PTP {X 66.600,Y -280.193,Z 129.598,A 103.371,B 90.000,C 0.000}
PTP {X 62.438,Y -262.681,Z 129.598,A 103.371,B 90.000,C 0.000}
PTP {X 62.202,Y -262.737,Z 133.786,A 103.319,B 90.000,C 0.000}
PTP {X 66.349,Y -280.253,Z 133.786,A 103.319,B 90.000,C 0.000}
WAIT SEC 2
RET=EKI_SetBool("oxy","torchState",TRUE)
RET = EKI_Send("oxy","torchState")
LIN {X 66.809,Y -282.199,Z 133.786,A 103.319,B 90.000,C 0.000} C_DIS
LIN {X 67.031,Y -282.147,Z 133.851,A 103.364,B 90.000,C 0.000} C_DIS
LIN {X 67.040,Y -282.145,Z 134.927,A 103.366,B 90.000,C 0.000} C_DIS
LIN {X 67.058,Y -282.140,Z 135.029,A 103.370,B 90.000,C 0.000} C_DIS
LIN {X 67.027,Y -282.148,Z 135.471,A 103.363,B 90.000,C 0.000} C_DIS
LIN {X 66.883,Y -282.182,Z 135.935,A 103.334,B 90.000,C 0.000} C_DIS
LIN {X 64.447,Y -282.742,Z 135.913,A 102.840,B 90.000,C 0.000} C_DIS
LIN {X 62.008,Y -283.292,Z 135.871,A 102.346,B 90.000,C 0.000} C_DIS
LIN {X 60.171,Y -283.689,Z 135.751,A 101.975,B 90.000,C 0.000} C_DIS
LIN {X 60.206,Y -283.682,Z 133.837,A 101.982,B 90.000,C 0.000} C_DIS
LIN {X 60.321,Y -283.657,Z 133.653,A 102.005,B 90.000,C 0.000} C_DIS
LIN {X 60.398,Y -283.641,Z 133.605,A 102.021,B 90.000,C 0.000} C_DIS
LIN {X 60.945,Y -283.524,Z 133.589,A 102.131,B 90.000,C 0.000} C_DIS
LIN {X 61.019,Y -283.508,Z 133.573,A 102.146,B 90.000,C 0.000} C_DIS
LIN {X 63.459,Y -282.971,Z 133.658,A 102.640,B 90.000,C 0.000} C_DIS
LIN {X 63.947,Y -282.862,Z 133.676,A 102.739,B 90.000,C 0.000} C_DIS
LIN {X 64.010,Y -282.847,Z 133.664,A 102.752,B 90.000,C 0.000} C_DIS
LIN {X 65.452,Y -282.517,Z 133.698,A 103.044,B 90.000,C 0.000} C_DIS
LIN {X 65.509,Y -282.504,Z 133.682,A 103.055,B 90.000,C 0.000} C_DIS
LIN {X 66.809,Y -282.199,Z 133.786,A 103.319,B 90.000,C 0.000} C_DIS
RET=EKI_SetBool("oxy","torchState",FALSE)
RET = EKI_Send("oxy","torchState")
PTP {X 66.349,Y -280.253,Z 133.786,A 103.319,B 90.000,C 0.000}
PTP {X 62.202,Y -262.737,Z 133.786,A 103.319,B 90.000,C 0.000}
PTP {X 62.126,Y -262.755,Z 137.889,A 103.303,B 90.000,C 0.000}
PTP {X 66.268,Y -280.272,Z 137.889,A 103.303,B 90.000,C 0.000}
WAIT SEC 2
RET=EKI_SetBool("oxy","torchState",TRUE)
RET = EKI_Send("oxy","torchState")
LIN {X 66.728,Y -282.219,Z 137.889,A 103.303,B 90.000,C 0.000} C_DIS
LIN {X 66.797,Y -282.202,Z 138.015,A 103.317,B 90.000,C 0.000} C_DIS
LIN {X 66.769,Y -282.209,Z 139.898,A 103.311,B 90.000,C 0.000} C_DIS
LIN {X 66.664,Y -282.234,Z 140.107,A 103.290,B 90.000,C 0.000} C_DIS
LIN {X 65.640,Y -282.474,Z 140.148,A 103.082,B 90.000,C 0.000} C_DIS
LIN {X 65.555,Y -282.493,Z 140.162,A 103.065,B 90.000,C 0.000} C_DIS
LIN {X 63.119,Y -283.046,Z 140.069,A 102.571,B 90.000,C 0.000} C_DIS
LIN {X 60.679,Y -283.581,Z 139.983,A 102.078,B 90.000,C 0.000} C_DIS
LIN {X 60.222,Y -283.678,Z 139.925,A 101.985,B 90.000,C 0.000} C_DIS
LIN {X 60.149,Y -283.694,Z 139.106,A 101.971,B 90.000,C 0.000} C_DIS
LIN {X 60.192,Y -283.685,Z 138.004,A 101.979,B 90.000,C 0.000} C_DIS
LIN {X 60.238,Y -283.675,Z 137.718,A 101.989,B 90.000,C 0.000} C_DIS
LIN {X 62.449,Y -283.196,Z 137.774,A 102.436,B 90.000,C 0.000} C_DIS
LIN {X 62.511,Y -283.183,Z 137.749,A 102.448,B 90.000,C 0.000} C_DIS
LIN {X 62.630,Y -283.156,Z 137.723,A 102.472,B 90.000,C 0.000} C_DIS
LIN {X 65.064,Y -282.605,Z 137.854,A 102.965,B 90.000,C 0.000} C_DIS
LIN {X 65.785,Y -282.440,Z 137.892,A 103.111,B 90.000,C 0.000} C_DIS
LIN {X 65.895,Y -282.414,Z 137.874,A 103.134,B 90.000,C 0.000} C_DIS
LIN {X 66.728,Y -282.219,Z 137.889,A 103.303,B 90.000,C 0.000} C_DIS
RET=EKI_SetBool("oxy","torchState",FALSE)
RET = EKI_Send("oxy","torchState")
PTP {X 66.268,Y -280.272,Z 137.889,A 103.303,B 90.000,C 0.000}
PTP {X 62.126,Y -262.755,Z 137.889,A 103.303,B 90.000,C 0.000}
PTP {X 63.167,Y -262.507,Z 145.772,A 103.530,B 90.000,C 0.000}
PTP {X 67.378,Y -280.008,Z 145.772,A 103.530,B 90.000,C 0.000}
WAIT SEC 2
RET=EKI_SetBool("oxy","torchState",TRUE)
RET = EKI_Send("oxy","torchState")
LIN {X 67.846,Y -281.952,Z 145.772,A 103.530,B 90.000,C 0.000} C_DIS
LIN {X 67.709,Y -281.985,Z 145.810,A 103.502,B 90.000,C 0.000} C_DIS
LIN {X 67.614,Y -282.008,Z 145.931,A 103.483,B 90.000,C 0.000} C_DIS
LIN {X 67.474,Y -282.041,Z 147.023,A 103.454,B 90.000,C 0.000} C_DIS
LIN {X 67.502,Y -282.035,Z 147.081,A 103.460,B 90.000,C 0.000} C_DIS
LIN {X 67.529,Y -282.028,Z 147.194,A 103.465,B 90.000,C 0.000} C_DIS
LIN {X 67.438,Y -282.050,Z 149.692,A 103.447,B 90.000,C 0.000} C_DIS
LIN {X 67.377,Y -282.064,Z 152.191,A 103.435,B 90.000,C 0.000} C_DIS
LIN {X 67.312,Y -282.080,Z 153.552,A 103.421,B 90.000,C 0.000} C_DIS
LIN {X 67.335,Y -282.075,Z 153.680,A 103.426,B 90.000,C 0.000} C_DIS
LIN {X 67.359,Y -282.069,Z 153.744,A 103.431,B 90.000,C 0.000} C_DIS
LIN {X 67.267,Y -282.091,Z 156.242,A 103.412,B 90.000,C 0.000} C_DIS
LIN {X 67.200,Y -282.107,Z 157.545,A 103.399,B 90.000,C 0.000} C_DIS
LIN {X 67.251,Y -282.094,Z 157.665,A 103.409,B 90.000,C 0.000} C_DIS
LIN {X 67.142,Y -282.120,Z 159.596,A 103.387,B 90.000,C 0.000} C_DIS
LIN {X 67.193,Y -282.108,Z 159.718,A 103.397,B 90.000,C 0.000} C_DIS
LIN {X 67.089,Y -282.133,Z 161.522,A 103.376,B 90.000,C 0.000} C_DIS
LIN {X 67.066,Y -282.138,Z 163.614,A 103.371,B 90.000,C 0.000} C_DIS
LIN {X 67.082,Y -282.135,Z 163.700,A 103.375,B 90.000,C 0.000} C_DIS
LIN {X 66.977,Y -282.160,Z 165.512,A 103.353,B 90.000,C 0.000} C_DIS
LIN {X 67.026,Y -282.148,Z 165.700,A 103.363,B 90.000,C 0.000} C_DIS
LIN {X 66.921,Y -282.173,Z 167.562,A 103.342,B 90.000,C 0.000} C_DIS
LIN {X 66.950,Y -282.166,Z 167.620,A 103.348,B 90.000,C 0.000} C_DIS
LIN {X 66.977,Y -282.160,Z 167.720,A 103.353,B 90.000,C 0.000} C_DIS
LIN {X 66.865,Y -282.186,Z 169.553,A 103.331,B 90.000,C 0.000} C_DIS
LIN {X 66.919,Y -282.173,Z 169.669,A 103.342,B 90.000,C 0.000} C_DIS
LIN {X 66.814,Y -282.198,Z 171.481,A 103.320,B 90.000,C 0.000} C_DIS
LIN {X 66.838,Y -282.193,Z 171.575,A 103.325,B 90.000,C 0.000} C_DIS
LIN {X 66.861,Y -282.187,Z 171.729,A 103.330,B 90.000,C 0.000} C_DIS
LIN {X 66.757,Y -282.212,Z 173.475,A 103.309,B 90.000,C 0.000} C_DIS
LIN {X 66.804,Y -282.201,Z 173.665,A 103.318,B 90.000,C 0.000} C_DIS
LIN {X 66.702,Y -282.225,Z 175.522,A 103.298,B 90.000,C 0.000} C_DIS
LIN {X 66.727,Y -282.219,Z 175.585,A 103.303,B 90.000,C 0.000} C_DIS
LIN {X 66.753,Y -282.213,Z 175.702,A 103.308,B 90.000,C 0.000} C_DIS
LIN {X 66.647,Y -282.238,Z 177.513,A 103.286,B 90.000,C 0.000} C_DIS
LIN {X 66.696,Y -282.226,Z 177.638,A 103.296,B 90.000,C 0.000} C_DIS
LIN {X 66.604,Y -282.248,Z 180.136,A 103.278,B 90.000,C 0.000} C_DIS
LIN {X 66.541,Y -282.263,Z 182.635,A 103.265,B 90.000,C 0.000} C_DIS
LIN {X 66.482,Y -282.277,Z 183.486,A 103.253,B 90.000,C 0.000} C_DIS
LIN {X 66.505,Y -282.271,Z 183.551,A 103.258,B 90.000,C 0.000} C_DIS
LIN {X 66.530,Y -282.265,Z 183.673,A 103.263,B 90.000,C 0.000} C_DIS
LIN {X 66.435,Y -282.288,Z 186.171,A 103.243,B 90.000,C 0.000} C_DIS
LIN {X 66.371,Y -282.303,Z 188.670,A 103.230,B 90.000,C 0.000} C_DIS
LIN {X 66.301,Y -282.319,Z 191.169,A 103.216,B 90.000,C 0.000} C_DIS
LIN {X 66.233,Y -282.335,Z 193.668,A 103.202,B 90.000,C 0.000} C_DIS
LIN {X 66.164,Y -282.351,Z 196.167,A 103.188,B 90.000,C 0.000} C_DIS
LIN {X 66.094,Y -282.368,Z 198.666,A 103.174,B 90.000,C 0.000} C_DIS
LIN {X 66.026,Y -282.384,Z 201.165,A 103.160,B 90.000,C 0.000} C_DIS
LIN {X 65.962,Y -282.399,Z 203.664,A 103.147,B 90.000,C 0.000} C_DIS
LIN {X 65.872,Y -282.420,Z 205.953,A 103.129,B 90.000,C 0.000} C_DIS
LIN {X 65.895,Y -282.414,Z 206.081,A 103.134,B 90.000,C 0.000} C_DIS
LIN {X 65.919,Y -282.409,Z 206.145,A 103.139,B 90.000,C 0.000} C_DIS
LIN {X 65.815,Y -282.433,Z 207.949,A 103.118,B 90.000,C 0.000} C_DIS
LIN {X 65.778,Y -282.442,Z 209.438,A 103.110,B 90.000,C 0.000} C_DIS
LIN {X 65.893,Y -282.415,Z 210.148,A 103.133,B 90.000,C 0.000} C_DIS
LIN {X 66.114,Y -282.363,Z 210.265,A 103.178,B 90.000,C 0.000} C_DIS
LIN {X 68.542,Y -281.784,Z 210.399,A 103.671,B 90.000,C 0.000} C_DIS
LIN {X 70.968,Y -281.181,Z 210.381,A 104.165,B 90.000,C 0.000} C_DIS
LIN {X 72.559,Y -280.776,Z 210.270,A 104.489,B 90.000,C 0.000} C_DIS
LIN {X 73.021,Y -280.656,Z 210.199,A 104.584,B 90.000,C 0.000} C_DIS
LIN {X 73.200,Y -280.610,Z 210.143,A 104.620,B 90.000,C 0.000} C_DIS
LIN {X 75.002,Y -280.133,Z 209.853,A 104.989,B 90.000,C 0.000} C_DIS
LIN {X 75.137,Y -280.097,Z 209.840,A 105.016,B 90.000,C 0.000} C_DIS
LIN {X 76.430,Y -279.747,Z 209.490,A 105.281,B 90.000,C 0.000} C_DIS
LIN {X 76.539,Y -279.717,Z 209.479,A 105.303,B 90.000,C 0.000} C_DIS
LIN {X 76.649,Y -279.687,Z 209.442,A 105.326,B 90.000,C 0.000} C_DIS
LIN {X 76.707,Y -279.671,Z 209.412,A 105.338,B 90.000,C 0.000} C_DIS
LIN {X 77.910,Y -279.338,Z 209.194,A 105.584,B 90.000,C 0.000} C_DIS
LIN {X 78.896,Y -279.062,Z 208.865,A 105.787,B 90.000,C 0.000} C_DIS
LIN {X 79.006,Y -279.031,Z 208.853,A 105.809,B 90.000,C 0.000} C_DIS
LIN {X 79.115,Y -279.000,Z 208.815,A 105.832,B 90.000,C 0.000} C_DIS
LIN {X 79.827,Y -278.797,Z 208.658,A 105.978,B 90.000,C 0.000} C_DIS
LIN {X 79.936,Y -278.766,Z 208.645,A 106.000,B 90.000,C 0.000} C_DIS
LIN {X 80.538,Y -278.592,Z 208.403,A 106.124,B 90.000,C 0.000} C_DIS
LIN {X 80.647,Y -278.561,Z 208.374,A 106.146,B 90.000,C 0.000} C_DIS
LIN {X 80.756,Y -278.529,Z 208.362,A 106.169,B 90.000,C 0.000} C_DIS
LIN {X 81.548,Y -278.298,Z 208.093,A 106.332,B 90.000,C 0.000} C_DIS
LIN {X 81.630,Y -278.274,Z 208.080,A 106.349,B 90.000,C 0.000} C_DIS
LIN {X 82.830,Y -277.919,Z 207.617,A 106.596,B 90.000,C 0.000} C_DIS
LIN {X 83.757,Y -277.641,Z 207.332,A 106.787,B 90.000,C 0.000} C_DIS
LIN {X 83.975,Y -277.576,Z 207.294,A 106.832,B 90.000,C 0.000} C_DIS
LIN {X 84.846,Y -277.311,Z 206.990,A 107.012,B 90.000,C 0.000} C_DIS
LIN {X 85.063,Y -277.244,Z 206.951,A 107.057,B 90.000,C 0.000} C_DIS
LIN {X 86.613,Y -276.764,Z 206.308,A 107.377,B 90.000,C 0.000} C_DIS
LIN {X 86.697,Y -276.737,Z 206.283,A 107.395,B 90.000,C 0.000} C_DIS
LIN {X 87.703,Y -276.420,Z 205.797,A 107.603,B 90.000,C 0.000} C_DIS
LIN {X 88.687,Y -276.106,Z 205.372,A 107.807,B 90.000,C 0.000} C_DIS
LIN {X 88.808,Y -276.067,Z 205.284,A 107.833,B 90.000,C 0.000} C_DIS
LIN {X 89.188,Y -275.945,Z 205.105,A 107.911,B 90.000,C 0.000} C_DIS
LIN {X 89.296,Y -275.910,Z 205.067,A 107.934,B 90.000,C 0.000} C_DIS
LIN {X 89.823,Y -275.739,Z 204.794,A 108.043,B 90.000,C 0.000} C_DIS
LIN {X 90.663,Y -275.464,Z 204.379,A 108.218,B 90.000,C 0.000} C_DIS
LIN {X 92.554,Y -274.834,Z 202.870,A 108.612,B 90.000,C 0.000} C_DIS
LIN {X 93.451,Y -274.530,Z 202.156,A 108.799,B 90.000,C 0.000} C_DIS
LIN {X 93.559,Y -274.494,Z 201.985,A 108.821,B 90.000,C 0.000} C_DIS
LIN {X 94.606,Y -274.134,Z 200.990,A 109.040,B 90.000,C 0.000} C_DIS
LIN {X 94.818,Y -274.061,Z 200.829,A 109.084,B 90.000,C 0.000} C_DIS
LIN {X 94.853,Y -274.049,Z 200.808,A 109.092,B 90.000,C 0.000} C_DIS
LIN {X 95.087,Y -273.968,Z 200.545,A 109.140,B 90.000,C 0.000} C_DIS
LIN {X 95.122,Y -273.956,Z 200.519,A 109.148,B 90.000,C 0.000} C_DIS
LIN {X 96.142,Y -273.600,Z 199.308,A 109.361,B 90.000,C 0.000} C_DIS
LIN {X 96.196,Y -273.581,Z 199.282,A 109.373,B 90.000,C 0.000} C_DIS
LIN {X 96.303,Y -273.543,Z 199.169,A 109.395,B 90.000,C 0.000} C_DIS
LIN {X 96.357,Y -273.524,Z 199.141,A 109.406,B 90.000,C 0.000} C_DIS
LIN {X 97.431,Y -273.143,Z 198.002,A 109.631,B 90.000,C 0.000} C_DIS
LIN {X 97.483,Y -273.125,Z 197.926,A 109.642,B 90.000,C 0.000} C_DIS
LIN {X 97.808,Y -273.008,Z 197.547,A 109.711,B 90.000,C 0.000} C_DIS
LIN {X 98.019,Y -272.933,Z 197.324,A 109.755,B 90.000,C 0.000} C_DIS
LIN {X 98.099,Y -272.904,Z 197.263,A 109.772,B 90.000,C 0.000} C_DIS
LIN {X 98.179,Y -272.875,Z 197.185,A 109.788,B 90.000,C 0.000} C_DIS
LIN {X 98.447,Y -272.779,Z 196.822,A 109.845,B 90.000,C 0.000} C_DIS
LIN {X 98.607,Y -272.721,Z 196.691,A 109.878,B 90.000,C 0.000} C_DIS
LIN {X 99.051,Y -272.560,Z 196.054,A 109.972,B 90.000,C 0.000} C_DIS
LIN {X 99.196,Y -272.507,Z 195.893,A 110.002,B 90.000,C 0.000} C_DIS
LIN {X 99.262,Y -272.483,Z 195.758,A 110.016,B 90.000,C 0.000} C_DIS
LIN {X 99.556,Y -272.376,Z 195.354,A 110.078,B 90.000,C 0.000} C_DIS
LIN {X 99.623,Y -272.351,Z 195.227,A 110.092,B 90.000,C 0.000} C_DIS
LIN {X 99.883,Y -272.256,Z 194.840,A 110.147,B 90.000,C 0.000} C_DIS
LIN {X 99.968,Y -272.225,Z 194.655,A 110.164,B 90.000,C 0.000} C_DIS
LIN {X 100.104,Y -272.175,Z 194.472,A 110.193,B 90.000,C 0.000} C_DIS
LIN {X 100.380,Y -272.073,Z 194.019,A 110.251,B 90.000,C 0.000} C_DIS
LIN {X 100.452,Y -272.047,Z 193.834,A 110.267,B 90.000,C 0.000} C_DIS
LIN {X 101.164,Y -271.783,Z 192.678,A 110.416,B 90.000,C 0.000} C_DIS
LIN {X 101.248,Y -271.751,Z 192.493,A 110.434,B 90.000,C 0.000} C_DIS
LIN {X 101.331,Y -271.721,Z 192.369,A 110.452,B 90.000,C 0.000} C_DIS
LIN {X 101.568,Y -271.632,Z 191.936,A 110.502,B 90.000,C 0.000} C_DIS
LIN {X 101.758,Y -271.561,Z 191.510,A 110.542,B 90.000,C 0.000} C_DIS
LIN {X 101.917,Y -271.501,Z 191.230,A 110.575,B 90.000,C 0.000} C_DIS
LIN {X 101.990,Y -271.474,Z 191.048,A 110.591,B 90.000,C 0.000} C_DIS
LIN {X 102.290,Y -271.361,Z 190.459,A 110.654,B 90.000,C 0.000} C_DIS
LIN {X 102.665,Y -271.219,Z 189.752,A 110.733,B 90.000,C 0.000} C_DIS
LIN {X 102.929,Y -271.119,Z 189.330,A 110.789,B 90.000,C 0.000} C_DIS
LIN {X 103.194,Y -271.018,Z 188.842,A 110.845,B 90.000,C 0.000} C_DIS
LIN {X 103.731,Y -270.813,Z 187.875,A 110.959,B 90.000,C 0.000} C_DIS
LIN {X 104.098,Y -270.673,Z 187.190,A 111.036,B 90.000,C 0.000} C_DIS
LIN {X 104.287,Y -270.600,Z 186.773,A 111.076,B 90.000,C 0.000} C_DIS
LIN {X 105.306,Y -270.205,Z 184.524,A 111.292,B 90.000,C 0.000} C_DIS
LIN {X 106.047,Y -269.915,Z 182.154,A 111.449,B 90.000,C 0.000} C_DIS
LIN {X 106.672,Y -269.668,Z 179.747,A 111.582,B 90.000,C 0.000} C_DIS
LIN {X 106.947,Y -269.560,Z 178.502,A 111.641,B 90.000,C 0.000} C_DIS
LIN {X 107.012,Y -269.534,Z 178.401,A 111.654,B 90.000,C 0.000} C_DIS
LIN {X 107.641,Y -269.283,Z 175.995,A 111.788,B 90.000,C 0.000} C_DIS
LIN {X 108.204,Y -269.057,Z 173.569,A 111.908,B 90.000,C 0.000} C_DIS
LIN {X 108.758,Y -268.834,Z 171.142,A 112.026,B 90.000,C 0.000} C_DIS
LIN {X 109.297,Y -268.615,Z 168.710,A 112.141,B 90.000,C 0.000} C_DIS
LIN {X 109.764,Y -268.425,Z 166.262,A 112.241,B 90.000,C 0.000} C_DIS
LIN {X 110.124,Y -268.277,Z 163.793,A 112.317,B 90.000,C 0.000} C_DIS
LIN {X 110.419,Y -268.156,Z 161.313,A 112.380,B 90.000,C 0.000} C_DIS
LIN {X 110.734,Y -268.026,Z 158.836,A 112.448,B 90.000,C 0.000} C_DIS
LIN {X 111.105,Y -267.873,Z 156.369,A 112.527,B 90.000,C 0.000} C_DIS
LIN {X 111.493,Y -267.711,Z 153.905,A 112.610,B 90.000,C 0.000} C_DIS
LIN {X 111.867,Y -267.555,Z 151.438,A 112.690,B 90.000,C 0.000} C_DIS
LIN {X 111.944,Y -267.523,Z 150.914,A 112.707,B 90.000,C 0.000} C_DIS
LIN {X 111.866,Y -267.556,Z 150.619,A 112.690,B 90.000,C 0.000} C_DIS
LIN {X 111.637,Y -267.651,Z 150.611,A 112.641,B 90.000,C 0.000} C_DIS
LIN {X 111.312,Y -267.787,Z 150.818,A 112.571,B 90.000,C 0.000} C_DIS
LIN {X 110.388,Y -268.169,Z 152.148,A 112.374,B 90.000,C 0.000} C_DIS
LIN {X 110.323,Y -268.196,Z 152.283,A 112.360,B 90.000,C 0.000} C_DIS
LIN {X 110.033,Y -268.315,Z 152.687,A 112.298,B 90.000,C 0.000} C_DIS
LIN {X 109.967,Y -268.342,Z 152.823,A 112.284,B 90.000,C 0.000} C_DIS
LIN {X 109.888,Y -268.374,Z 152.884,A 112.267,B 90.000,C 0.000} C_DIS
LIN {X 109.809,Y -268.406,Z 152.967,A 112.250,B 90.000,C 0.000} C_DIS
LIN {X 109.230,Y -268.643,Z 153.798,A 112.127,B 90.000,C 0.000} C_DIS
LIN {X 108.492,Y -268.942,Z 154.770,A 111.969,B 90.000,C 0.000} C_DIS
LIN {X 108.452,Y -268.958,Z 154.799,A 111.961,B 90.000,C 0.000} C_DIS
LIN {X 108.344,Y -269.001,Z 154.853,A 111.938,B 90.000,C 0.000} C_DIS
LIN {X 108.308,Y -269.015,Z 154.932,A 111.930,B 90.000,C 0.000} C_DIS
LIN {X 107.700,Y -269.260,Z 155.660,A 111.801,B 90.000,C 0.000} C_DIS
LIN {X 107.466,Y -269.353,Z 155.857,A 111.751,B 90.000,C 0.000} C_DIS
LIN {X 107.013,Y -269.534,Z 156.459,A 111.654,B 90.000,C 0.000} C_DIS
LIN {X 106.880,Y -269.586,Z 156.582,A 111.626,B 90.000,C 0.000} C_DIS
LIN {X 106.245,Y -269.837,Z 157.322,A 111.492,B 90.000,C 0.000} C_DIS
LIN {X 106.166,Y -269.868,Z 157.383,A 111.475,B 90.000,C 0.000} C_DIS
LIN {X 105.958,Y -269.950,Z 157.606,A 111.430,B 90.000,C 0.000} C_DIS
LIN {X 104.629,Y -270.468,Z 159.264,A 111.149,B 90.000,C 0.000} C_DIS
LIN {X 104.523,Y -270.509,Z 159.301,A 111.126,B 90.000,C 0.000} C_DIS
LIN {X 104.416,Y -270.550,Z 159.484,A 111.104,B 90.000,C 0.000} C_DIS
LIN {X 104.204,Y -270.632,Z 159.654,A 111.059,B 90.000,C 0.000} C_DIS
LIN {X 104.098,Y -270.673,Z 159.837,A 111.036,B 90.000,C 0.000} C_DIS
LIN {X 104.045,Y -270.693,Z 159.853,A 111.025,B 90.000,C 0.000} C_DIS
LIN {X 103.992,Y -270.713,Z 159.879,A 111.014,B 90.000,C 0.000} C_DIS
LIN {X 103.939,Y -270.734,Z 159.939,A 111.003,B 90.000,C 0.000} C_DIS
LIN {X 102.916,Y -271.124,Z 160.863,A 110.786,B 90.000,C 0.000} C_DIS
LIN {X 102.761,Y -271.183,Z 160.963,A 110.753,B 90.000,C 0.000} C_DIS
LIN {X 101.118,Y -271.800,Z 162.344,A 110.407,B 90.000,C 0.000} C_DIS
LIN {X 101.011,Y -271.840,Z 162.370,A 110.384,B 90.000,C 0.000} C_DIS
LIN {X 99.164,Y -272.519,Z 163.912,A 109.996,B 90.000,C 0.000} C_DIS
LIN {X 97.915,Y -272.970,Z 164.946,A 109.733,B 90.000,C 0.000} C_DIS
LIN {X 96.893,Y -273.334,Z 165.569,A 109.519,B 90.000,C 0.000} C_DIS
LIN {X 96.679,Y -273.410,Z 165.629,A 109.474,B 90.000,C 0.000} C_DIS
LIN {X 96.303,Y -273.543,Z 165.812,A 109.395,B 90.000,C 0.000} C_DIS
LIN {X 96.088,Y -273.618,Z 165.859,A 109.350,B 90.000,C 0.000} C_DIS
LIN {X 95.713,Y -273.750,Z 166.028,A 109.271,B 90.000,C 0.000} C_DIS
LIN {X 95.498,Y -273.825,Z 166.067,A 109.226,B 90.000,C 0.000} C_DIS
LIN {X 94.630,Y -274.126,Z 166.389,A 109.045,B 90.000,C 0.000} C_DIS
LIN {X 93.080,Y -274.656,Z 166.682,A 108.721,B 90.000,C 0.000} C_DIS
LIN {X 93.001,Y -274.683,Z 166.718,A 108.705,B 90.000,C 0.000} C_DIS
LIN {X 92.699,Y -274.785,Z 166.760,A 108.642,B 90.000,C 0.000} C_DIS
LIN {X 92.626,Y -274.810,Z 166.790,A 108.627,B 90.000,C 0.000} C_DIS
LIN {X 91.350,Y -275.236,Z 166.921,A 108.361,B 90.000,C 0.000} C_DIS
LIN {X 90.329,Y -275.573,Z 166.912,A 108.148,B 90.000,C 0.000} C_DIS
LIN {X 90.217,Y -275.610,Z 166.966,A 108.125,B 90.000,C 0.000} C_DIS
LIN {X 87.844,Y -276.375,Z 166.775,A 107.633,B 90.000,C 0.000} C_DIS
LIN {X 87.119,Y -276.605,Z 166.677,A 107.482,B 90.000,C 0.000} C_DIS
LIN {X 84.832,Y -277.315,Z 165.959,A 107.009,B 90.000,C 0.000} C_DIS
LIN {X 82.557,Y -278.000,Z 165.182,A 106.540,B 90.000,C 0.000} C_DIS
LIN {X 80.348,Y -278.647,Z 164.206,A 106.085,B 90.000,C 0.000} C_DIS
LIN {X 79.018,Y -279.027,Z 163.487,A 105.812,B 90.000,C 0.000} C_DIS
LIN {X 78.732,Y -279.108,Z 163.351,A 105.753,B 90.000,C 0.000} C_DIS
LIN {X 77.702,Y -279.397,Z 162.449,A 105.542,B 90.000,C 0.000} C_DIS
LIN {X 77.129,Y -279.555,Z 161.793,A 105.424,B 90.000,C 0.000} C_DIS
LIN {X 76.943,Y -279.606,Z 161.674,A 105.386,B 90.000,C 0.000} C_DIS
LIN {X 75.441,Y -280.015,Z 160.166,A 105.078,B 90.000,C 0.000} C_DIS
LIN {X 74.857,Y -280.172,Z 159.269,A 104.959,B 90.000,C 0.000} C_DIS
LIN {X 74.741,Y -280.203,Z 158.962,A 104.935,B 90.000,C 0.000} C_DIS
LIN {X 74.452,Y -280.280,Z 158.354,A 104.876,B 90.000,C 0.000} C_DIS
LIN {X 74.402,Y -280.293,Z 158.289,A 104.866,B 90.000,C 0.000} C_DIS
LIN {X 74.351,Y -280.307,Z 158.061,A 104.855,B 90.000,C 0.000} C_DIS
LIN {X 74.147,Y -280.361,Z 157.610,A 104.814,B 90.000,C 0.000} C_DIS
LIN {X 74.129,Y -280.366,Z 157.525,A 104.810,B 90.000,C 0.000} C_DIS
LIN {X 73.627,Y -280.498,Z 156.152,A 104.708,B 90.000,C 0.000} C_DIS
LIN {X 73.751,Y -280.465,Z 156.076,A 104.733,B 90.000,C 0.000} C_DIS
LIN {X 74.007,Y -280.398,Z 156.226,A 104.785,B 90.000,C 0.000} C_DIS
LIN {X 74.243,Y -280.336,Z 156.451,A 104.833,B 90.000,C 0.000} C_DIS
LIN {X 74.452,Y -280.280,Z 156.750,A 104.876,B 90.000,C 0.000} C_DIS
LIN {X 74.516,Y -280.263,Z 156.810,A 104.889,B 90.000,C 0.000} C_DIS
LIN {X 74.546,Y -280.255,Z 156.845,A 104.895,B 90.000,C 0.000} C_DIS
LIN {X 75.606,Y -279.971,Z 158.296,A 105.112,B 90.000,C 0.000} C_DIS
LIN {X 76.808,Y -279.644,Z 159.541,A 105.358,B 90.000,C 0.000} C_DIS
LIN {X 77.227,Y -279.528,Z 159.825,A 105.444,B 90.000,C 0.000} C_DIS
LIN {X 77.394,Y -279.482,Z 159.967,A 105.479,B 90.000,C 0.000} C_DIS
LIN {X 77.606,Y -279.423,Z 160.109,A 105.522,B 90.000,C 0.000} C_DIS
LIN {X 77.691,Y -279.399,Z 160.195,A 105.539,B 90.000,C 0.000} C_DIS
LIN {X 77.748,Y -279.384,Z 160.280,A 105.551,B 90.000,C 0.000} C_DIS
LIN {X 78.369,Y -279.210,Z 160.753,A 105.679,B 90.000,C 0.000} C_DIS
LIN {X 78.515,Y -279.169,Z 160.906,A 105.708,B 90.000,C 0.000} C_DIS
LIN {X 78.639,Y -279.134,Z 160.964,A 105.734,B 90.000,C 0.000} C_DIS
LIN {X 79.151,Y -278.990,Z 161.333,A 105.839,B 90.000,C 0.000} C_DIS
LIN {X 80.846,Y -278.503,Z 162.328,A 106.187,B 90.000,C 0.000} C_DIS
LIN {X 80.920,Y -278.481,Z 162.383,A 106.203,B 90.000,C 0.000} C_DIS
LIN {X 81.866,Y -278.205,Z 162.810,A 106.397,B 90.000,C 0.000} C_DIS
LIN {X 82.273,Y -278.085,Z 163.047,A 106.481,B 90.000,C 0.000} C_DIS
LIN {X 82.447,Y -278.033,Z 163.125,A 106.517,B 90.000,C 0.000} C_DIS
LIN {X 84.030,Y -277.559,Z 163.866,A 106.843,B 90.000,C 0.000} C_DIS
LIN {X 86.363,Y -276.840,Z 164.401,A 107.326,B 90.000,C 0.000} C_DIS
LIN {X 87.752,Y -276.405,Z 164.640,A 107.613,B 90.000,C 0.000} C_DIS
LIN {X 90.131,Y -275.637,Z 164.640,A 108.107,B 90.000,C 0.000} C_DIS
LIN {X 91.761,Y -275.100,Z 164.513,A 108.446,B 90.000,C 0.000} C_DIS
LIN {X 91.836,Y -275.075,Z 164.484,A 108.462,B 90.000,C 0.000} C_DIS
LIN {X 93.171,Y -274.626,Z 164.264,A 108.740,B 90.000,C 0.000} C_DIS
LIN {X 93.292,Y -274.584,Z 164.199,A 108.766,B 90.000,C 0.000} C_DIS
LIN {X 93.380,Y -274.555,Z 164.172,A 108.784,B 90.000,C 0.000} C_DIS
LIN {X 93.777,Y -274.419,Z 164.099,A 108.867,B 90.000,C 0.000} C_DIS
LIN {X 95.444,Y -273.844,Z 163.519,A 109.215,B 90.000,C 0.000} C_DIS
LIN {X 95.511,Y -273.820,Z 163.468,A 109.229,B 90.000,C 0.000} C_DIS
LIN {X 96.402,Y -273.508,Z 162.997,A 109.416,B 90.000,C 0.000} C_DIS
LIN {X 96.469,Y -273.485,Z 162.986,A 109.430,B 90.000,C 0.000} C_DIS
LIN {X 96.989,Y -273.301,Z 162.727,A 109.539,B 90.000,C 0.000} C_DIS
LIN {X 97.342,Y -273.175,Z 162.596,A 109.613,B 90.000,C 0.000} C_DIS
LIN {X 97.376,Y -273.163,Z 162.565,A 109.620,B 90.000,C 0.000} C_DIS
LIN {X 97.469,Y -273.129,Z 162.499,A 109.640,B 90.000,C 0.000} C_DIS
LIN {X 97.978,Y -272.947,Z 162.272,A 109.746,B 90.000,C 0.000} C_DIS
LIN {X 98.458,Y -272.775,Z 161.955,A 109.847,B 90.000,C 0.000} C_DIS
LIN {X 98.643,Y -272.708,Z 161.852,A 109.886,B 90.000,C 0.000} C_DIS
LIN {X 98.926,Y -272.605,Z 161.646,A 109.945,B 90.000,C 0.000} C_DIS
LIN {X 99.013,Y -272.574,Z 161.546,A 109.964,B 90.000,C 0.000} C_DIS
LIN {X 99.249,Y -272.488,Z 161.371,A 110.013,B 90.000,C 0.000} C_DIS
LIN {X 99.946,Y -272.233,Z 160.721,A 110.160,B 90.000,C 0.000} C_DIS
LIN {X 100.102,Y -272.176,Z 160.521,A 110.193,B 90.000,C 0.000} C_DIS
LIN {X 101.700,Y -271.583,Z 159.072,A 110.529,B 90.000,C 0.000} C_DIS
LIN {X 101.811,Y -271.541,Z 158.998,A 110.553,B 90.000,C 0.000} C_DIS
LIN {X 103.534,Y -270.889,Z 157.309,A 110.917,B 90.000,C 0.000} C_DIS
LIN {X 104.204,Y -270.632,Z 156.381,A 111.059,B 90.000,C 0.000} C_DIS
LIN {X 104.257,Y -270.611,Z 156.326,A 111.070,B 90.000,C 0.000} C_DIS
LIN {X 104.310,Y -270.591,Z 156.302,A 111.081,B 90.000,C 0.000} C_DIS
LIN {X 104.894,Y -270.365,Z 155.561,A 111.205,B 90.000,C 0.000} C_DIS
LIN {X 104.947,Y -270.344,Z 155.529,A 111.216,B 90.000,C 0.000} C_DIS
LIN {X 105.000,Y -270.324,Z 155.509,A 111.227,B 90.000,C 0.000} C_DIS
LIN {X 106.587,Y -269.702,Z 153.680,A 111.564,B 90.000,C 0.000} C_DIS
LIN {X 107.541,Y -269.323,Z 152.538,A 111.767,B 90.000,C 0.000} C_DIS
LIN {X 107.594,Y -269.302,Z 152.514,A 111.778,B 90.000,C 0.000} C_DIS
LIN {X 107.647,Y -269.281,Z 152.480,A 111.789,B 90.000,C 0.000} C_DIS
LIN {X 108.333,Y -269.005,Z 151.590,A 111.936,B 90.000,C 0.000} C_DIS
LIN {X 108.492,Y -268.942,Z 151.457,A 111.969,B 90.000,C 0.000} C_DIS
LIN {X 108.558,Y -268.915,Z 151.315,A 111.983,B 90.000,C 0.000} C_DIS
LIN {X 109.190,Y -268.659,Z 150.547,A 112.118,B 90.000,C 0.000} C_DIS
LIN {X 109.335,Y -268.600,Z 150.320,A 112.149,B 90.000,C 0.000} C_DIS
LIN {X 109.493,Y -268.535,Z 150.142,A 112.183,B 90.000,C 0.000} C_DIS
LIN {X 110.275,Y -268.215,Z 149.144,A 112.350,B 90.000,C 0.000} C_DIS
LIN {X 110.407,Y -268.161,Z 149.054,A 112.378,B 90.000,C 0.000} C_DIS
LIN {X 110.757,Y -268.017,Z 148.530,A 112.453,B 90.000,C 0.000} C_DIS
LIN {X 110.809,Y -267.995,Z 148.474,A 112.464,B 90.000,C 0.000} C_DIS
LIN {X 110.862,Y -267.973,Z 148.450,A 112.475,B 90.000,C 0.000} C_DIS
LIN {X 111.177,Y -267.843,Z 147.995,A 112.543,B 90.000,C 0.000} C_DIS
LIN {X 111.226,Y -267.822,Z 147.960,A 112.553,B 90.000,C 0.000} C_DIS
LIN {X 111.308,Y -267.788,Z 147.878,A 112.571,B 90.000,C 0.000} C_DIS
LIN {X 111.391,Y -267.754,Z 147.763,A 112.588,B 90.000,C 0.000} C_DIS
LIN {X 112.204,Y -267.414,Z 146.500,A 112.762,B 90.000,C 0.000} C_DIS
LIN {X 113.158,Y -267.012,Z 144.224,A 112.967,B 90.000,C 0.000} C_DIS
LIN {X 113.967,Y -266.667,Z 141.884,A 113.141,B 90.000,C 0.000} C_DIS
LIN {X 114.668,Y -266.367,Z 139.503,A 113.291,B 90.000,C 0.000} C_DIS
LIN {X 115.419,Y -266.042,Z 137.141,A 113.453,B 90.000,C 0.000} C_DIS
LIN {X 116.181,Y -265.710,Z 134.783,A 113.617,B 90.000,C 0.000} C_DIS
LIN {X 116.912,Y -265.390,Z 132.414,A 113.775,B 90.000,C 0.000} C_DIS
LIN {X 117.615,Y -265.079,Z 130.035,A 113.927,B 90.000,C 0.000} C_DIS
LIN {X 118.323,Y -264.763,Z 127.659,A 114.080,B 90.000,C 0.000} C_DIS
LIN {X 119.096,Y -264.416,Z 125.307,A 114.247,B 90.000,C 0.000} C_DIS
LIN {X 119.968,Y -264.022,Z 122.997,A 114.436,B 90.000,C 0.000} C_DIS
LIN {X 120.871,Y -263.610,Z 120.703,A 114.632,B 90.000,C 0.000} C_DIS
LIN {X 121.669,Y -263.242,Z 118.620,A 114.806,B 90.000,C 0.000} C_DIS
LIN {X 121.984,Y -263.097,Z 117.906,A 114.875,B 90.000,C 0.000} C_DIS
LIN {X 122.322,Y -262.940,Z 117.160,A 114.948,B 90.000,C 0.000} C_DIS
LIN {X 123.186,Y -262.536,Z 114.849,A 115.137,B 90.000,C 0.000} C_DIS
LIN {X 124.147,Y -262.083,Z 112.587,A 115.347,B 90.000,C 0.000} C_DIS
LIN {X 124.998,Y -261.678,Z 110.271,A 115.533,B 90.000,C 0.000} C_DIS
LIN {X 125.720,Y -261.332,Z 107.903,A 115.691,B 90.000,C 0.000} C_DIS
LIN {X 126.434,Y -260.988,Z 105.532,A 115.848,B 90.000,C 0.000} C_DIS
LIN {X 127.087,Y -260.670,Z 103.140,A 115.991,B 90.000,C 0.000} C_DIS
LIN {X 127.896,Y -260.274,Z 100.808,A 116.169,B 90.000,C 0.000} C_DIS
LIN {X 128.611,Y -259.921,Z 98.438,A 116.327,B 90.000,C 0.000} C_DIS
LIN {X 129.304,Y -259.577,Z 96.061,A 116.479,B 90.000,C 0.000} C_DIS
LIN {X 129.860,Y -259.300,Z 93.826,A 116.602,B 90.000,C 0.000} C_DIS
LIN {X 129.878,Y -259.291,Z 91.326,A 116.606,B 90.000,C 0.000} C_DIS
LIN {X 129.664,Y -259.398,Z 90.184,A 116.559,B 90.000,C 0.000} C_DIS
LIN {X 129.650,Y -259.405,Z 90.071,A 116.556,B 90.000,C 0.000} C_DIS
LIN {X 129.441,Y -259.509,Z 89.331,A 116.510,B 90.000,C 0.000} C_DIS
LIN {X 129.431,Y -259.514,Z 89.217,A 116.507,B 90.000,C 0.000} C_DIS
LIN {X 129.405,Y -259.527,Z 89.103,A 116.502,B 90.000,C 0.000} C_DIS
LIN {X 128.834,Y -259.811,Z 87.432,A 116.376,B 90.000,C 0.000} C_DIS
LIN {X 128.444,Y -260.004,Z 86.844,A 116.290,B 90.000,C 0.000} C_DIS
LIN {X 127.967,Y -260.239,Z 86.374,A 116.185,B 90.000,C 0.000} C_DIS
LIN {X 127.426,Y -260.505,Z 85.860,A 116.066,B 90.000,C 0.000} C_DIS
LIN {X 127.035,Y -260.695,Z 85.660,A 115.980,B 90.000,C 0.000} C_DIS
LIN {X 126.875,Y -260.773,Z 85.655,A 115.945,B 90.000,C 0.000} C_DIS
LIN {X 126.821,Y -260.799,Z 85.825,A 115.933,B 90.000,C 0.000} C_DIS
LIN {X 126.949,Y -260.737,Z 87.081,A 115.961,B 90.000,C 0.000} C_DIS
LIN {X 126.899,Y -260.762,Z 88.211,A 115.950,B 90.000,C 0.000} C_DIS
LIN {X 126.851,Y -260.785,Z 88.284,A 115.939,B 90.000,C 0.000} C_DIS
LIN {X 126.585,Y -260.914,Z 89.160,A 115.881,B 90.000,C 0.000} C_DIS
LIN {X 126.308,Y -261.049,Z 89.772,A 115.820,B 90.000,C 0.000} C_DIS
LIN {X 125.305,Y -261.531,Z 91.315,A 115.600,B 90.000,C 0.000} C_DIS
LIN {X 125.177,Y -261.593,Z 91.436,A 115.572,B 90.000,C 0.000} C_DIS
LIN {X 125.049,Y -261.654,Z 91.588,A 115.544,B 90.000,C 0.000} C_DIS
LIN {X 125.005,Y -261.675,Z 91.664,A 115.534,B 90.000,C 0.000} C_DIS
LIN {X 124.484,Y -261.923,Z 92.243,A 115.420,B 90.000,C 0.000} C_DIS
LIN {X 124.450,Y -261.939,Z 92.272,A 115.413,B 90.000,C 0.000} C_DIS
LIN {X 124.227,Y -262.045,Z 92.529,A 115.364,B 90.000,C 0.000} C_DIS
LIN {X 124.185,Y -262.065,Z 92.552,A 115.355,B 90.000,C 0.000} C_DIS
LIN {X 124.069,Y -262.120,Z 92.639,A 115.330,B 90.000,C 0.000} C_DIS
LIN {X 123.241,Y -262.510,Z 93.541,A 115.149,B 90.000,C 0.000} C_DIS
LIN {X 123.198,Y -262.531,Z 93.617,A 115.139,B 90.000,C 0.000} C_DIS
LIN {X 122.885,Y -262.677,Z 93.996,A 115.071,B 90.000,C 0.000} C_DIS
LIN {X 122.682,Y -262.772,Z 94.220,A 115.027,B 90.000,C 0.000} C_DIS
LIN {X 122.527,Y -262.844,Z 94.352,A 114.993,B 90.000,C 0.000} C_DIS
LIN {X 122.373,Y -262.916,Z 94.622,A 114.959,B 90.000,C 0.000} C_DIS
LIN {X 122.173,Y -263.009,Z 94.883,A 114.916,B 90.000,C 0.000} C_DIS
LIN {X 121.988,Y -263.095,Z 95.305,A 114.876,B 90.000,C 0.000} C_DIS
LIN {X 121.316,Y -263.406,Z 97.693,A 114.729,B 90.000,C 0.000} C_DIS
LIN {X 120.723,Y -263.678,Z 100.106,A 114.600,B 90.000,C 0.000} C_DIS
LIN {X 120.099,Y -263.962,Z 102.510,A 114.465,B 90.000,C 0.000} C_DIS
LIN {X 119.449,Y -264.257,Z 104.906,A 114.324,B 90.000,C 0.000} C_DIS
LIN {X 118.758,Y -264.569,Z 107.288,A 114.174,B 90.000,C 0.000} C_DIS
LIN {X 118.141,Y -264.845,Z 109.695,A 114.041,B 90.000,C 0.000} C_DIS
LIN {X 117.546,Y -265.109,Z 112.108,A 113.912,B 90.000,C 0.000} C_DIS
LIN {X 116.921,Y -265.385,Z 114.513,A 113.777,B 90.000,C 0.000} C_DIS
LIN {X 116.310,Y -265.654,Z 116.922,A 113.645,B 90.000,C 0.000} C_DIS
LIN {X 115.717,Y -265.913,Z 119.337,A 113.517,B 90.000,C 0.000} C_DIS
LIN {X 115.102,Y -266.180,Z 121.746,A 113.385,B 90.000,C 0.000} C_DIS
LIN {X 114.399,Y -266.482,Z 124.126,A 113.234,B 90.000,C 0.000} C_DIS
LIN {X 114.213,Y -266.562,Z 124.720,A 113.193,B 90.000,C 0.000} C_DIS
LIN {X 113.366,Y -266.924,Z 127.044,A 113.012,B 90.000,C 0.000} C_DIS
LIN {X 112.561,Y -267.264,Z 129.387,A 112.839,B 90.000,C 0.000} C_DIS
LIN {X 112.070,Y -267.470,Z 130.688,A 112.734,B 90.000,C 0.000} C_DIS
LIN {X 111.841,Y -267.566,Z 131.334,A 112.685,B 90.000,C 0.000} C_DIS
LIN {X 111.282,Y -267.799,Z 132.578,A 112.565,B 90.000,C 0.000} C_DIS
LIN {X 111.125,Y -267.864,Z 132.858,A 112.531,B 90.000,C 0.000} C_DIS
LIN {X 110.938,Y -267.942,Z 133.276,A 112.491,B 90.000,C 0.000} C_DIS
LIN {X 110.599,Y -268.082,Z 133.946,A 112.419,B 90.000,C 0.000} C_DIS
LIN {X 110.283,Y -268.212,Z 134.508,A 112.351,B 90.000,C 0.000} C_DIS
LIN {X 110.211,Y -268.242,Z 134.690,A 112.336,B 90.000,C 0.000} C_DIS
LIN {X 110.102,Y -268.286,Z 134.893,A 112.313,B 90.000,C 0.000} C_DIS
LIN {X 109.622,Y -268.483,Z 135.713,A 112.210,B 90.000,C 0.000} C_DIS
LIN {X 109.441,Y -268.557,Z 136.075,A 112.172,B 90.000,C 0.000} C_DIS
LIN {X 109.016,Y -268.729,Z 136.782,A 112.081,B 90.000,C 0.000} C_DIS
LIN {X 108.912,Y -268.772,Z 137.010,A 112.059,B 90.000,C 0.000} C_DIS
LIN {X 108.807,Y -268.814,Z 137.138,A 112.036,B 90.000,C 0.000} C_DIS
LIN {X 108.333,Y -269.005,Z 137.975,A 111.936,B 90.000,C 0.000} C_DIS
LIN {X 108.201,Y -269.059,Z 138.148,A 111.907,B 90.000,C 0.000} C_DIS
LIN {X 108.069,Y -269.112,Z 138.288,A 111.879,B 90.000,C 0.000} C_DIS
LIN {X 107.990,Y -269.143,Z 138.412,A 111.862,B 90.000,C 0.000} C_DIS
LIN {X 106.748,Y -269.638,Z 140.143,A 111.598,B 90.000,C 0.000} C_DIS
LIN {X 106.589,Y -269.701,Z 140.309,A 111.565,B 90.000,C 0.000} C_DIS
LIN {X 105.742,Y -270.034,Z 141.399,A 111.385,B 90.000,C 0.000} C_DIS
LIN {X 105.636,Y -270.076,Z 141.440,A 111.362,B 90.000,C 0.000} C_DIS
LIN {X 104.845,Y -270.384,Z 142.405,A 111.194,B 90.000,C 0.000} C_DIS
LIN {X 104.682,Y -270.447,Z 142.529,A 111.160,B 90.000,C 0.000} C_DIS
LIN {X 103.017,Y -271.086,Z 144.281,A 110.808,B 90.000,C 0.000} C_DIS
LIN {X 102.397,Y -271.321,Z 144.786,A 110.677,B 90.000,C 0.000} C_DIS
LIN {X 102.165,Y -271.408,Z 145.050,A 110.628,B 90.000,C 0.000} C_DIS
LIN {X 102.062,Y -271.447,Z 145.146,A 110.606,B 90.000,C 0.000} C_DIS
LIN {X 101.805,Y -271.543,Z 145.341,A 110.552,B 90.000,C 0.000} C_DIS
LIN {X 101.647,Y -271.602,Z 145.513,A 110.518,B 90.000,C 0.000} C_DIS
LIN {X 101.598,Y -271.621,Z 145.532,A 110.508,B 90.000,C 0.000} C_DIS
LIN {X 101.225,Y -271.760,Z 145.842,A 110.429,B 90.000,C 0.000} C_DIS
LIN {X 101.145,Y -271.790,Z 145.886,A 110.412,B 90.000,C 0.000} C_DIS
LIN {X 101.065,Y -271.820,Z 145.946,A 110.396,B 90.000,C 0.000} C_DIS
LIN {X 101.011,Y -271.840,Z 145.971,A 110.384,B 90.000,C 0.000} C_DIS
LIN {X 100.958,Y -271.859,Z 145.987,A 110.373,B 90.000,C 0.000} C_DIS
LIN {X 100.544,Y -272.013,Z 146.332,A 110.286,B 90.000,C 0.000} C_DIS
LIN {X 98.406,Y -272.794,Z 147.364,A 109.836,B 90.000,C 0.000} C_DIS
LIN {X 98.286,Y -272.837,Z 147.419,A 109.811,B 90.000,C 0.000} C_DIS
LIN {X 98.072,Y -272.914,Z 147.462,A 109.766,B 90.000,C 0.000} C_DIS
LIN {X 97.215,Y -273.220,Z 147.783,A 109.586,B 90.000,C 0.000} C_DIS
LIN {X 94.960,Y -274.012,Z 148.209,A 109.114,B 90.000,C 0.000} C_DIS
LIN {X 94.887,Y -274.037,Z 148.242,A 109.099,B 90.000,C 0.000} C_DIS
LIN {X 93.736,Y -274.433,Z 148.353,A 108.858,B 90.000,C 0.000} C_DIS
LIN {X 93.615,Y -274.474,Z 148.381,A 108.833,B 90.000,C 0.000} C_DIS
LIN {X 93.544,Y -274.499,Z 148.413,A 108.818,B 90.000,C 0.000} C_DIS
LIN {X 92.128,Y -274.977,Z 148.594,A 108.523,B 90.000,C 0.000} C_DIS
LIN {X 92.052,Y -275.003,Z 148.623,A 108.507,B 90.000,C 0.000} C_DIS
LIN {X 91.703,Y -275.119,Z 148.671,A 108.434,B 90.000,C 0.000} C_DIS
LIN {X 91.624,Y -275.146,Z 148.704,A 108.418,B 90.000,C 0.000} C_DIS
LIN {X 89.260,Y -275.921,Z 148.950,A 107.926,B 90.000,C 0.000} C_DIS
LIN {X 87.823,Y -276.382,Z 149.039,A 107.628,B 90.000,C 0.000} C_DIS
LIN {X 86.924,Y -276.666,Z 148.991,A 107.442,B 90.000,C 0.000} C_DIS
LIN {X 86.215,Y -276.888,Z 149.011,A 107.295,B 90.000,C 0.000} C_DIS
LIN {X 86.133,Y -276.913,Z 149.043,A 107.278,B 90.000,C 0.000} C_DIS
LIN {X 84.093,Y -277.540,Z 149.020,A 106.856,B 90.000,C 0.000} C_DIS
LIN {X 84.023,Y -277.561,Z 149.039,A 106.842,B 90.000,C 0.000} C_DIS
LIN {X 81.633,Y -278.272,Z 148.853,A 106.349,B 90.000,C 0.000} C_DIS
LIN {X 80.016,Y -278.743,Z 148.672,A 106.017,B 90.000,C 0.000} C_DIS
LIN {X 77.655,Y -279.408,Z 148.190,A 105.532,B 90.000,C 0.000} C_DIS
LIN {X 75.284,Y -280.057,Z 147.737,A 105.046,B 90.000,C 0.000} C_DIS
LIN {X 72.953,Y -280.674,Z 147.075,A 104.570,B 90.000,C 0.000} C_DIS
LIN {X 70.603,Y -281.272,Z 146.468,A 104.091,B 90.000,C 0.000} C_DIS
LIN {X 68.246,Y -281.855,Z 145.874,A 103.611,B 90.000,C 0.000} C_DIS
LIN {X 67.846,Y -281.952,Z 145.772,A 103.530,B 90.000,C 0.000} C_DIS
RET=EKI_SetBool("oxy","torchState",FALSE)
RET = EKI_Send("oxy","torchState")
PTP {X 67.378,Y -280.008,Z 145.772,A 103.530,B 90.000,C 0.000}
PTP {X 63.167,Y -262.507,Z 145.772,A 103.530,B 90.000,C 0.000}
PTP {X 54.029,Y -264.539,Z 140.807,A 101.543,B 90.000,C 0.000}
PTP {X 57.631,Y -282.175,Z 140.807,A 101.543,B 90.000,C 0.000}
WAIT SEC 2
RET=EKI_SetBool("oxy","torchState",TRUE)
RET = EKI_Send("oxy","torchState")
LIN {X 58.031,Y -284.135,Z 140.807,A 101.543,B 90.000,C 0.000} C_DIS
LIN {X 57.952,Y -284.151,Z 140.920,A 101.527,B 90.000,C 0.000} C_DIS
LIN {X 56.798,Y -284.383,Z 141.343,A 101.295,B 90.000,C 0.000} C_DIS
LIN {X 56.716,Y -284.400,Z 141.360,A 101.278,B 90.000,C 0.000} C_DIS
LIN {X 56.274,Y -284.488,Z 141.560,A 101.189,B 90.000,C 0.000} C_DIS
LIN {X 56.050,Y -284.532,Z 141.620,A 101.144,B 90.000,C 0.000} C_DIS
LIN {X 55.771,Y -284.587,Z 141.795,A 101.088,B 90.000,C 0.000} C_DIS
LIN {X 55.045,Y -284.728,Z 142.141,A 100.942,B 90.000,C 0.000} C_DIS
LIN {X 54.318,Y -284.868,Z 142.358,A 100.795,B 90.000,C 0.000} C_DIS
LIN {X 54.207,Y -284.889,Z 142.416,A 100.773,B 90.000,C 0.000} C_DIS
LIN {X 53.928,Y -284.942,Z 142.469,A 100.717,B 90.000,C 0.000} C_DIS
LIN {X 53.868,Y -284.953,Z 142.498,A 100.705,B 90.000,C 0.000} C_DIS
LIN {X 51.477,Y -285.395,Z 143.080,A 100.225,B 90.000,C 0.000} C_DIS
LIN {X 51.410,Y -285.407,Z 143.089,A 100.211,B 90.000,C 0.000} C_DIS
LIN {X 50.178,Y -285.626,Z 143.446,A 99.964,B 90.000,C 0.000} C_DIS
LIN {X 50.065,Y -285.646,Z 143.455,A 99.941,B 90.000,C 0.000} C_DIS
LIN {X 49.508,Y -285.743,Z 143.594,A 99.829,B 90.000,C 0.000} C_DIS
LIN {X 47.175,Y -286.137,Z 144.043,A 99.362,B 90.000,C 0.000} C_DIS
LIN {X 47.093,Y -286.151,Z 144.071,A 99.346,B 90.000,C 0.000} C_DIS
LIN {X 46.756,Y -286.206,Z 144.107,A 99.278,B 90.000,C 0.000} C_DIS
LIN {X 46.573,Y -286.236,Z 144.162,A 99.242,B 90.000,C 0.000} C_DIS
LIN {X 44.104,Y -286.621,Z 144.225,A 98.748,B 90.000,C 0.000} C_DIS
LIN {X 41.633,Y -286.996,Z 144.183,A 98.254,B 90.000,C 0.000} C_DIS
LIN {X 39.168,Y -287.343,Z 143.947,A 97.762,B 90.000,C 0.000} C_DIS
LIN {X 38.358,Y -287.452,Z 143.787,A 97.601,B 90.000,C 0.000} C_DIS
LIN {X 37.820,Y -287.523,Z 143.608,A 97.494,B 90.000,C 0.000} C_DIS
LIN {X 36.113,Y -287.743,Z 142.757,A 97.154,B 90.000,C 0.000} C_DIS
LIN {X 35.787,Y -287.783,Z 142.549,A 97.089,B 90.000,C 0.000} C_DIS
LIN {X 35.492,Y -287.820,Z 142.413,A 97.030,B 90.000,C 0.000} C_DIS
LIN {X 35.210,Y -287.855,Z 142.188,A 96.974,B 90.000,C 0.000} C_DIS
LIN {X 34.615,Y -287.927,Z 141.789,A 96.855,B 90.000,C 0.000} C_DIS
LIN {X 34.505,Y -287.940,Z 141.675,A 96.833,B 90.000,C 0.000} C_DIS
LIN {X 34.193,Y -287.977,Z 141.446,A 96.771,B 90.000,C 0.000} C_DIS
LIN {X 33.060,Y -288.109,Z 140.309,A 96.546,B 90.000,C 0.000} C_DIS
LIN {X 33.025,Y -288.113,Z 140.267,A 96.539,B 90.000,C 0.000} C_DIS
LIN {X 32.978,Y -288.119,Z 140.157,A 96.530,B 90.000,C 0.000} C_DIS
LIN {X 32.871,Y -288.131,Z 140.123,A 96.508,B 90.000,C 0.000} C_DIS
LIN {X 32.837,Y -288.135,Z 140.100,A 96.502,B 90.000,C 0.000} C_DIS
LIN {X 31.492,Y -288.285,Z 138.219,A 96.234,B 90.000,C 0.000} C_DIS
LIN {X 31.026,Y -288.336,Z 137.351,A 96.142,B 90.000,C 0.000} C_DIS
LIN {X 30.971,Y -288.341,Z 137.298,A 96.131,B 90.000,C 0.000} C_DIS
LIN {X 30.848,Y -288.355,Z 136.881,A 96.106,B 90.000,C 0.000} C_DIS
LIN {X 30.801,Y -288.360,Z 136.839,A 96.097,B 90.000,C 0.000} C_DIS
LIN {X 30.744,Y -288.366,Z 136.774,A 96.086,B 90.000,C 0.000} C_DIS
LIN {X 30.428,Y -288.399,Z 136.014,A 96.023,B 90.000,C 0.000} C_DIS
LIN {X 29.888,Y -288.456,Z 134.335,A 95.916,B 90.000,C 0.000} C_DIS
LIN {X 29.879,Y -288.457,Z 134.222,A 95.914,B 90.000,C 0.000} C_DIS
LIN {X 29.799,Y -288.465,Z 133.994,A 95.898,B 90.000,C 0.000} C_DIS
LIN {X 29.499,Y -288.496,Z 131.832,A 95.838,B 90.000,C 0.000} C_DIS
LIN {X 29.472,Y -288.499,Z 130.906,A 95.833,B 90.000,C 0.000} C_DIS
LIN {X 29.574,Y -288.488,Z 129.828,A 95.853,B 90.000,C 0.000} C_DIS
LIN {X 29.669,Y -288.478,Z 129.529,A 95.872,B 90.000,C 0.000} C_DIS
LIN {X 29.949,Y -288.449,Z 129.101,A 95.928,B 90.000,C 0.000} C_DIS
LIN {X 31.197,Y -288.317,Z 127.665,A 96.176,B 90.000,C 0.000} C_DIS
LIN {X 31.230,Y -288.314,Z 127.636,A 96.182,B 90.000,C 0.000} C_DIS
LIN {X 31.373,Y -288.298,Z 127.573,A 96.210,B 90.000,C 0.000} C_DIS
LIN {X 31.480,Y -288.286,Z 127.407,A 96.232,B 90.000,C 0.000} C_DIS
LIN {X 31.536,Y -288.280,Z 127.366,A 96.243,B 90.000,C 0.000} C_DIS
LIN {X 31.593,Y -288.274,Z 127.341,A 96.254,B 90.000,C 0.000} C_DIS
LIN {X 31.649,Y -288.268,Z 127.280,A 96.266,B 90.000,C 0.000} C_DIS
LIN {X 32.803,Y -288.139,Z 126.355,A 96.495,B 90.000,C 0.000} C_DIS
LIN {X 32.837,Y -288.135,Z 126.323,A 96.502,B 90.000,C 0.000} C_DIS
LIN {X 32.922,Y -288.125,Z 126.256,A 96.518,B 90.000,C 0.000} C_DIS
LIN {X 33.006,Y -288.116,Z 126.212,A 96.535,B 90.000,C 0.000} C_DIS
LIN {X 33.402,Y -288.070,Z 125.902,A 96.614,B 90.000,C 0.000} C_DIS
LIN {X 33.515,Y -288.057,Z 125.870,A 96.636,B 90.000,C 0.000} C_DIS
LIN {X 33.911,Y -288.011,Z 125.560,A 96.715,B 90.000,C 0.000} C_DIS
LIN {X 34.476,Y -287.943,Z 125.245,A 96.828,B 90.000,C 0.000} C_DIS
LIN {X 34.871,Y -287.896,Z 124.935,A 96.906,B 90.000,C 0.000} C_DIS
LIN {X 34.928,Y -287.889,Z 124.919,A 96.917,B 90.000,C 0.000} C_DIS
LIN {X 34.984,Y -287.882,Z 124.894,A 96.929,B 90.000,C 0.000} C_DIS
LIN {X 35.067,Y -287.872,Z 124.834,A 96.945,B 90.000,C 0.000} C_DIS
LIN {X 36.326,Y -287.716,Z 124.172,A 97.196,B 90.000,C 0.000} C_DIS
LIN {X 36.650,Y -287.675,Z 124.036,A 97.260,B 90.000,C 0.000} C_DIS
LIN {X 36.738,Y -287.664,Z 124.011,A 97.278,B 90.000,C 0.000} C_DIS
LIN {X 36.791,Y -287.657,Z 123.984,A 97.288,B 90.000,C 0.000} C_DIS
LIN {X 36.862,Y -287.648,Z 123.923,A 97.303,B 90.000,C 0.000} C_DIS
LIN {X 37.439,Y -287.573,Z 123.696,A 97.418,B 90.000,C 0.000} C_DIS
LIN {X 37.708,Y -287.538,Z 123.551,A 97.471,B 90.000,C 0.000} C_DIS
LIN {X 39.554,Y -287.290,Z 122.899,A 97.839,B 90.000,C 0.000} C_DIS
LIN {X 39.667,Y -287.274,Z 122.883,A 97.862,B 90.000,C 0.000} C_DIS
LIN {X 39.893,Y -287.243,Z 122.802,A 97.907,B 90.000,C 0.000} C_DIS
LIN {X 40.005,Y -287.227,Z 122.792,A 97.929,B 90.000,C 0.000} C_DIS
LIN {X 41.019,Y -287.084,Z 122.495,A 98.132,B 90.000,C 0.000} C_DIS
LIN {X 41.132,Y -287.068,Z 122.485,A 98.154,B 90.000,C 0.000} C_DIS
LIN {X 41.692,Y -286.987,Z 122.346,A 98.266,B 90.000,C 0.000} C_DIS
LIN {X 44.021,Y -286.639,Z 121.908,A 98.731,B 90.000,C 0.000} C_DIS
LIN {X 44.115,Y -286.625,Z 121.877,A 98.750,B 90.000,C 0.000} C_DIS
LIN {X 44.283,Y -286.599,Z 121.847,A 98.784,B 90.000,C 0.000} C_DIS
LIN {X 44.452,Y -286.573,Z 121.837,A 98.817,B 90.000,C 0.000} C_DIS
LIN {X 44.663,Y -286.540,Z 121.782,A 98.859,B 90.000,C 0.000} C_DIS
LIN {X 47.036,Y -286.160,Z 121.630,A 99.334,B 90.000,C 0.000} C_DIS
LIN {X 47.093,Y -286.151,Z 121.620,A 99.346,B 90.000,C 0.000} C_DIS
LIN {X 49.550,Y -285.735,Z 121.825,A 99.838,B 90.000,C 0.000} C_DIS
LIN {X 51.967,Y -285.304,Z 122.294,A 100.323,B 90.000,C 0.000} C_DIS
LIN {X 53.003,Y -285.115,Z 122.536,A 100.531,B 90.000,C 0.000} C_DIS
LIN {X 55.265,Y -284.685,Z 123.511,A 100.986,B 90.000,C 0.000} C_DIS
LIN {X 57.307,Y -284.281,Z 124.663,A 101.397,B 90.000,C 0.000} C_DIS
LIN {X 57.362,Y -284.270,Z 124.720,A 101.408,B 90.000,C 0.000} C_DIS
LIN {X 57.381,Y -284.266,Z 124.777,A 101.412,B 90.000,C 0.000} C_DIS
LIN {X 58.185,Y -284.103,Z 125.630,A 101.574,B 90.000,C 0.000} C_DIS
LIN {X 58.198,Y -284.100,Z 125.687,A 101.577,B 90.000,C 0.000} C_DIS
LIN {X 58.223,Y -284.095,Z 125.744,A 101.582,B 90.000,C 0.000} C_DIS
LIN {X 58.332,Y -284.073,Z 125.915,A 101.604,B 90.000,C 0.000} C_DIS
LIN {X 58.354,Y -284.068,Z 126.029,A 101.608,B 90.000,C 0.000} C_DIS
LIN {X 58.433,Y -284.052,Z 126.256,A 101.624,B 90.000,C 0.000} C_DIS
LIN {X 58.442,Y -284.050,Z 126.370,A 101.626,B 90.000,C 0.000} C_DIS
LIN {X 58.730,Y -283.991,Z 127.367,A 101.684,B 90.000,C 0.000} C_DIS
LIN {X 58.744,Y -283.988,Z 127.508,A 101.687,B 90.000,C 0.000} C_DIS
LIN {X 58.813,Y -283.974,Z 127.731,A 101.701,B 90.000,C 0.000} C_DIS
LIN {X 58.865,Y -283.963,Z 130.230,A 101.711,B 90.000,C 0.000} C_DIS
LIN {X 58.751,Y -283.987,Z 132.727,A 101.688,B 90.000,C 0.000} C_DIS
LIN {X 58.700,Y -283.997,Z 133.482,A 101.678,B 90.000,C 0.000} C_DIS
LIN {X 58.721,Y -283.993,Z 133.539,A 101.682,B 90.000,C 0.000} C_DIS
LIN {X 58.750,Y -283.987,Z 133.667,A 101.688,B 90.000,C 0.000} C_DIS
LIN {X 58.641,Y -284.009,Z 134.966,A 101.666,B 90.000,C 0.000} C_DIS
LIN {X 58.674,Y -284.002,Z 135.018,A 101.673,B 90.000,C 0.000} C_DIS
LIN {X 58.700,Y -283.997,Z 135.118,A 101.678,B 90.000,C 0.000} C_DIS
LIN {X 58.515,Y -284.035,Z 137.611,A 101.641,B 90.000,C 0.000} C_DIS
LIN {X 58.157,Y -284.109,Z 140.084,A 101.569,B 90.000,C 0.000} C_DIS
LIN {X 58.031,Y -284.135,Z 140.807,A 101.543,B 90.000,C 0.000} C_DIS
RET=EKI_SetBool("oxy","torchState",FALSE)
RET = EKI_Send("oxy","torchState")
PTP {X 57.631,Y -282.175,Z 140.807,A 101.543,B 90.000,C 0.000}
PTP {X 54.029,Y -264.539,Z 140.807,A 101.543,B 90.000,C 0.000}
PTP {X 63.996,Y -262.306,Z 71.409,A 103.711,B 90.000,C 0.000}
PTP {X 68.262,Y -279.793,Z 71.409,A 103.711,B 90.000,C 0.000}
WAIT SEC 2
RET=EKI_SetBool("oxy","torchState",TRUE)
RET = EKI_Send("oxy","torchState")
LIN {X 68.736,Y -281.736,Z 71.409,A 103.711,B 90.000,C 0.000} C_DIS
LIN {X 68.662,Y -281.754,Z 71.361,A 103.696,B 90.000,C 0.000} C_DIS
LIN {X 67.868,Y -281.947,Z 70.584,A 103.534,B 90.000,C 0.000} C_DIS
LIN {X 67.748,Y -281.975,Z 70.498,A 103.510,B 90.000,C 0.000} C_DIS
LIN {X 67.695,Y -281.988,Z 70.441,A 103.499,B 90.000,C 0.000} C_DIS
LIN {X 67.681,Y -281.992,Z 70.385,A 103.496,B 90.000,C 0.000} C_DIS
LIN {X 65.248,Y -282.555,Z 70.293,A 103.003,B 90.000,C 0.000} C_DIS
LIN {X 63.166,Y -283.037,Z 70.214,A 102.581,B 90.000,C 0.000} C_DIS
LIN {X 62.122,Y -283.268,Z 71.105,A 102.369,B 90.000,C 0.000} C_DIS
LIN {X 62.080,Y -283.277,Z 71.181,A 102.361,B 90.000,C 0.000} C_DIS
LIN {X 60.156,Y -283.692,Z 72.723,A 101.972,B 90.000,C 0.000} C_DIS
LIN {X 58.533,Y -284.032,Z 74.026,A 101.644,B 90.000,C 0.000} C_DIS
LIN {X 57.051,Y -284.333,Z 75.221,A 101.346,B 90.000,C 0.000} C_DIS
LIN {X 56.164,Y -284.509,Z 76.131,A 101.167,B 90.000,C 0.000} C_DIS
LIN {X 56.048,Y -284.532,Z 76.302,A 101.144,B 90.000,C 0.000} C_DIS
LIN {X 55.922,Y -284.557,Z 76.360,A 101.118,B 90.000,C 0.000} C_DIS
LIN {X 54.872,Y -284.761,Z 77.185,A 100.907,B 90.000,C 0.000} C_DIS
LIN {X 54.670,Y -284.800,Z 77.418,A 100.866,B 90.000,C 0.000} C_DIS
LIN {X 53.309,Y -285.058,Z 78.635,A 100.593,B 90.000,C 0.000} C_DIS
LIN {X 52.529,Y -285.203,Z 79.301,A 100.436,B 90.000,C 0.000} C_DIS
LIN {X 52.482,Y -285.212,Z 79.374,A 100.426,B 90.000,C 0.000} C_DIS
LIN {X 51.158,Y -285.452,Z 80.703,A 100.160,B 90.000,C 0.000} C_DIS
LIN {X 51.074,Y -285.467,Z 80.816,A 100.144,B 90.000,C 0.000} C_DIS
LIN {X 50.907,Y -285.497,Z 81.137,A 100.110,B 90.000,C 0.000} C_DIS
LIN {X 50.963,Y -285.487,Z 81.339,A 100.121,B 90.000,C 0.000} C_DIS
LIN {X 51.127,Y -285.458,Z 81.518,A 100.154,B 90.000,C 0.000} C_DIS
LIN {X 51.578,Y -285.376,Z 81.707,A 100.245,B 90.000,C 0.000} C_DIS
LIN {X 51.690,Y -285.356,Z 81.780,A 100.267,B 90.000,C 0.000} C_DIS
LIN {X 51.802,Y -285.336,Z 81.767,A 100.290,B 90.000,C 0.000} C_DIS
LIN {X 53.420,Y -285.037,Z 81.904,A 100.615,B 90.000,C 0.000} C_DIS
LIN {X 53.480,Y -285.026,Z 81.875,A 100.627,B 90.000,C 0.000} C_DIS
LIN {X 53.578,Y -285.008,Z 81.849,A 100.647,B 90.000,C 0.000} C_DIS
LIN {X 56.032,Y -284.534,Z 81.925,A 101.140,B 90.000,C 0.000} C_DIS
LIN {X 57.043,Y -284.335,Z 81.955,A 101.344,B 90.000,C 0.000} C_DIS
LIN {X 57.120,Y -284.319,Z 81.934,A 101.360,B 90.000,C 0.000} C_DIS
LIN {X 57.668,Y -284.208,Z 81.923,A 101.470,B 90.000,C 0.000} C_DIS
LIN {X 57.788,Y -284.184,Z 81.909,A 101.494,B 90.000,C 0.000} C_DIS
LIN {X 60.233,Y -283.674,Z 82.001,A 101.988,B 90.000,C 0.000} C_DIS
LIN {X 62.676,Y -283.145,Z 82.061,A 102.481,B 90.000,C 0.000} C_DIS
LIN {X 63.996,Y -282.851,Z 82.129,A 102.749,B 90.000,C 0.000} C_DIS
LIN {X 64.121,Y -282.822,Z 82.106,A 102.774,B 90.000,C 0.000} C_DIS
LIN {X 64.183,Y -282.808,Z 82.081,A 102.787,B 90.000,C 0.000} C_DIS
LIN {X 65.941,Y -282.404,Z 82.187,A 103.143,B 90.000,C 0.000} C_DIS
LIN {X 66.061,Y -282.375,Z 82.163,A 103.167,B 90.000,C 0.000} C_DIS
LIN {X 66.123,Y -282.361,Z 82.138,A 103.180,B 90.000,C 0.000} C_DIS
LIN {X 68.553,Y -281.780,Z 82.233,A 103.674,B 90.000,C 0.000} C_DIS
LIN {X 69.831,Y -281.467,Z 82.303,A 103.934,B 90.000,C 0.000} C_DIS
LIN {X 69.959,Y -281.435,Z 82.279,A 103.960,B 90.000,C 0.000} C_DIS
LIN {X 70.048,Y -281.413,Z 82.250,A 103.978,B 90.000,C 0.000} C_DIS
LIN {X 71.808,Y -280.969,Z 82.361,A 104.336,B 90.000,C 0.000} C_DIS
LIN {X 71.926,Y -280.939,Z 82.309,A 104.360,B 90.000,C 0.000} C_DIS
LIN {X 73.672,Y -280.486,Z 82.415,A 104.717,B 90.000,C 0.000} C_DIS
LIN {X 73.792,Y -280.455,Z 82.390,A 104.741,B 90.000,C 0.000} C_DIS
LIN {X 73.849,Y -280.440,Z 82.362,A 104.753,B 90.000,C 0.000} C_DIS
LIN {X 76.261,Y -279.792,Z 82.467,A 105.246,B 90.000,C 0.000} C_DIS
LIN {X 77.522,Y -279.446,Z 82.529,A 105.505,B 90.000,C 0.000} C_DIS
LIN {X 77.581,Y -279.430,Z 82.513,A 105.517,B 90.000,C 0.000} C_DIS
LIN {X 78.061,Y -279.296,Z 82.533,A 105.615,B 90.000,C 0.000} C_DIS
LIN {X 78.129,Y -279.277,Z 82.505,A 105.629,B 90.000,C 0.000} C_DIS
LIN {X 78.253,Y -279.243,Z 82.479,A 105.655,B 90.000,C 0.000} C_DIS
LIN {X 78.575,Y -279.152,Z 82.469,A 105.721,B 90.000,C 0.000} C_DIS
LIN {X 78.857,Y -279.073,Z 82.364,A 105.779,B 90.000,C 0.000} C_DIS
LIN {X 78.998,Y -279.033,Z 82.006,A 105.807,B 90.000,C 0.000} C_DIS
LIN {X 78.997,Y -279.033,Z 81.707,A 105.807,B 90.000,C 0.000} C_DIS
LIN {X 78.951,Y -279.046,Z 81.623,A 105.798,B 90.000,C 0.000} C_DIS
LIN {X 78.403,Y -279.201,Z 80.898,A 105.685,B 90.000,C 0.000} C_DIS
LIN {X 78.239,Y -279.247,Z 80.798,A 105.652,B 90.000,C 0.000} C_DIS
LIN {X 76.550,Y -279.713,Z 79.015,A 105.306,B 90.000,C 0.000} C_DIS
LIN {X 75.377,Y -280.033,Z 77.781,A 105.065,B 90.000,C 0.000} C_DIS
LIN {X 75.348,Y -280.040,Z 77.744,A 105.060,B 90.000,C 0.000} C_DIS
LIN {X 75.100,Y -280.107,Z 77.497,A 105.009,B 90.000,C 0.000} C_DIS
LIN {X 75.081,Y -280.112,Z 77.444,A 105.005,B 90.000,C 0.000} C_DIS
LIN {X 75.002,Y -280.133,Z 77.355,A 104.989,B 90.000,C 0.000} C_DIS
LIN {X 74.507,Y -280.266,Z 76.988,A 104.887,B 90.000,C 0.000} C_DIS
LIN {X 74.305,Y -280.319,Z 76.832,A 104.846,B 90.000,C 0.000} C_DIS
LIN {X 73.792,Y -280.455,Z 76.131,A 104.741,B 90.000,C 0.000} C_DIS
LIN {X 73.681,Y -280.484,Z 76.045,A 104.719,B 90.000,C 0.000} C_DIS
LIN {X 73.601,Y -280.505,Z 75.956,A 104.702,B 90.000,C 0.000} C_DIS
LIN {X 73.576,Y -280.511,Z 75.904,A 104.697,B 90.000,C 0.000} C_DIS
LIN {X 72.071,Y -280.902,Z 74.538,A 104.390,B 90.000,C 0.000} C_DIS
LIN {X 72.057,Y -280.905,Z 74.481,A 104.387,B 90.000,C 0.000} C_DIS
LIN {X 72.003,Y -280.919,Z 74.424,A 104.376,B 90.000,C 0.000} C_DIS
LIN {X 71.025,Y -281.168,Z 73.514,A 104.177,B 90.000,C 0.000} C_DIS
LIN {X 69.208,Y -281.621,Z 71.858,A 103.807,B 90.000,C 0.000} C_DIS
LIN {X 69.105,Y -281.646,Z 71.752,A 103.786,B 90.000,C 0.000} C_DIS
LIN {X 68.736,Y -281.736,Z 71.409,A 103.711,B 90.000,C 0.000} C_DIS
RET=EKI_SetBool("oxy","torchState",FALSE)
RET = EKI_Send("oxy","torchState")
PTP {X 68.262,Y -279.793,Z 71.409,A 103.711,B 90.000,C 0.000}
PTP {X 63.996,Y -262.306,Z 71.409,A 103.711,B 90.000,C 0.000}
PTP {X 181.822,Y -199.601,Z 91.692,A 132.331,B 90.000,C 0.000}
PTP {X 193.944,Y -212.908,Z 91.692,A 132.331,B 90.000,C 0.000}
WAIT SEC 2
RET=EKI_SetBool("oxy","torchState",TRUE)
RET = EKI_Send("oxy","torchState")
LIN {X 195.290,Y -214.387,Z 91.692,A 132.331,B 90.000,C 0.000} C_DIS
LIN {X 195.329,Y -214.352,Z 91.529,A 132.341,B 90.000,C 0.000} C_DIS
LIN {X 195.367,Y -214.317,Z 91.497,A 132.352,B 90.000,C 0.000} C_DIS
LIN {X 195.382,Y -214.303,Z 91.419,A 132.356,B 90.000,C 0.000} C_DIS
LIN {X 195.457,Y -214.235,Z 91.222,A 132.376,B 90.000,C 0.000} C_DIS
LIN {X 195.632,Y -214.075,Z 90.971,A 132.423,B 90.000,C 0.000} C_DIS
LIN {X 195.835,Y -213.889,Z 90.754,A 132.477,B 90.000,C 0.000} C_DIS
LIN {X 195.994,Y -213.743,Z 90.662,A 132.520,B 90.000,C 0.000} C_DIS
LIN {X 196.089,Y -213.656,Z 90.641,A 132.545,B 90.000,C 0.000} C_DIS
LIN {X 196.129,Y -213.620,Z 90.590,A 132.556,B 90.000,C 0.000} C_DIS
LIN {X 196.302,Y -213.461,Z 90.537,A 132.602,B 90.000,C 0.000} C_DIS
LIN {X 197.231,Y -212.603,Z 90.537,A 132.852,B 90.000,C 0.000} C_DIS
LIN {X 197.403,Y -212.443,Z 90.590,A 132.898,B 90.000,C 0.000} C_DIS
LIN {X 197.449,Y -212.400,Z 90.641,A 132.911,B 90.000,C 0.000} C_DIS
LIN {X 197.674,Y -212.191,Z 90.684,A 132.971,B 90.000,C 0.000} C_DIS
LIN {X 197.767,Y -212.104,Z 90.786,A 132.997,B 90.000,C 0.000} C_DIS
LIN {X 197.991,Y -211.896,Z 90.828,A 133.057,B 90.000,C 0.000} C_DIS
LIN {X 198.037,Y -211.852,Z 90.879,A 133.070,B 90.000,C 0.000} C_DIS
LIN {X 198.099,Y -211.794,Z 90.930,A 133.086,B 90.000,C 0.000} C_DIS
LIN {X 198.397,Y -211.515,Z 90.973,A 133.167,B 90.000,C 0.000} C_DIS
LIN {X 198.459,Y -211.457,Z 91.024,A 133.184,B 90.000,C 0.000} C_DIS
LIN {X 198.505,Y -211.413,Z 91.075,A 133.196,B 90.000,C 0.000} C_DIS
LIN {X 198.729,Y -211.204,Z 91.117,A 133.257,B 90.000,C 0.000} C_DIS
LIN {X 198.775,Y -211.160,Z 91.168,A 133.270,B 90.000,C 0.000} C_DIS
LIN {X 198.837,Y -211.102,Z 91.219,A 133.286,B 90.000,C 0.000} C_DIS
LIN {X 199.134,Y -210.822,Z 91.262,A 133.367,B 90.000,C 0.000} C_DIS
LIN {X 199.196,Y -210.763,Z 91.313,A 133.384,B 90.000,C 0.000} C_DIS
LIN {X 199.242,Y -210.719,Z 91.364,A 133.396,B 90.000,C 0.000} C_DIS
LIN {X 199.464,Y -210.509,Z 91.406,A 133.457,B 90.000,C 0.000} C_DIS
LIN {X 199.510,Y -210.465,Z 91.457,A 133.469,B 90.000,C 0.000} C_DIS
LIN {X 199.572,Y -210.407,Z 91.508,A 133.486,B 90.000,C 0.000} C_DIS
LIN {X 199.868,Y -210.126,Z 91.551,A 133.567,B 90.000,C 0.000} C_DIS
LIN {X 199.930,Y -210.067,Z 91.602,A 133.584,B 90.000,C 0.000} C_DIS
LIN {X 199.975,Y -210.024,Z 91.676,A 133.596,B 90.000,C 0.000} C_DIS
LIN {X 200.086,Y -209.918,Z 91.668,A 133.626,B 90.000,C 0.000} C_DIS
LIN {X 200.223,Y -209.788,Z 91.591,A 133.664,B 90.000,C 0.000} C_DIS
LIN {X 200.890,Y -209.149,Z 90.871,A 133.846,B 90.000,C 0.000} C_DIS
LIN {X 201.056,Y -208.989,Z 90.764,A 133.892,B 90.000,C 0.000} C_DIS
LIN {X 201.210,Y -208.840,Z 90.560,A 133.934,B 90.000,C 0.000} C_DIS
LIN {X 201.298,Y -208.756,Z 90.518,A 133.958,B 90.000,C 0.000} C_DIS
LIN {X 201.363,Y -208.693,Z 90.497,A 133.976,B 90.000,C 0.000} C_DIS
LIN {X 201.421,Y -208.637,Z 90.394,A 133.992,B 90.000,C 0.000} C_DIS
LIN {X 201.568,Y -208.496,Z 90.352,A 134.032,B 90.000,C 0.000} C_DIS
LIN {X 201.598,Y -208.466,Z 90.301,A 134.040,B 90.000,C 0.000} C_DIS
LIN {X 201.644,Y -208.422,Z 90.250,A 134.053,B 90.000,C 0.000} C_DIS
LIN {X 201.864,Y -208.209,Z 90.207,A 134.114,B 90.000,C 0.000} C_DIS
LIN {X 201.955,Y -208.120,Z 90.105,A 134.139,B 90.000,C 0.000} C_DIS
LIN {X 202.175,Y -207.907,Z 90.063,A 134.199,B 90.000,C 0.000} C_DIS
LIN {X 202.221,Y -207.862,Z 90.012,A 134.212,B 90.000,C 0.000} C_DIS
LIN {X 202.297,Y -207.788,Z 89.961,A 134.233,B 90.000,C 0.000} C_DIS
LIN {X 202.662,Y -207.432,Z 89.918,A 134.334,B 90.000,C 0.000} C_DIS
LIN {X 202.738,Y -207.358,Z 89.867,A 134.355,B 90.000,C 0.000} C_DIS
LIN {X 202.932,Y -207.168,Z 89.814,A 134.408,B 90.000,C 0.000} C_DIS
LIN {X 203.987,Y -206.129,Z 89.814,A 134.701,B 90.000,C 0.000} C_DIS
LIN {X 204.180,Y -205.938,Z 89.867,A 134.754,B 90.000,C 0.000} C_DIS
LIN {X 204.240,Y -205.878,Z 89.918,A 134.771,B 90.000,C 0.000} C_DIS
LIN {X 204.530,Y -205.591,Z 89.961,A 134.852,B 90.000,C 0.000} C_DIS
LIN {X 204.590,Y -205.531,Z 90.012,A 134.869,B 90.000,C 0.000} C_DIS
LIN {X 204.635,Y -205.486,Z 90.063,A 134.881,B 90.000,C 0.000} C_DIS
LIN {X 204.852,Y -205.270,Z 90.105,A 134.942,B 90.000,C 0.000} C_DIS
LIN {X 204.942,Y -205.180,Z 90.207,A 134.967,B 90.000,C 0.000} C_DIS
LIN {X 205.159,Y -204.963,Z 90.250,A 135.027,B 90.000,C 0.000} C_DIS
LIN {X 205.204,Y -204.918,Z 90.301,A 135.040,B 90.000,C 0.000} C_DIS
LIN {X 205.234,Y -204.888,Z 90.352,A 135.048,B 90.000,C 0.000} C_DIS
LIN {X 205.378,Y -204.744,Z 90.394,A 135.089,B 90.000,C 0.000} C_DIS
LIN {X 205.438,Y -204.683,Z 90.497,A 135.105,B 90.000,C 0.000} C_DIS
LIN {X 205.582,Y -204.539,Z 90.539,A 135.146,B 90.000,C 0.000} C_DIS
LIN {X 205.612,Y -204.509,Z 90.590,A 135.154,B 90.000,C 0.000} C_DIS
LIN {X 205.636,Y -204.485,Z 90.641,A 135.161,B 90.000,C 0.000} C_DIS
LIN {X 205.693,Y -204.427,Z 90.662,A 135.177,B 90.000,C 0.000} C_DIS
LIN {X 205.793,Y -204.327,Z 90.726,A 135.205,B 90.000,C 0.000} C_DIS
LIN {X 206.278,Y -203.837,Z 91.263,A 135.341,B 90.000,C 0.000} C_DIS
LIN {X 206.816,Y -203.290,Z 92.039,A 135.493,B 90.000,C 0.000} C_DIS
LIN {X 207.034,Y -203.069,Z 92.469,A 135.554,B 90.000,C 0.000} C_DIS
LIN {X 207.105,Y -202.996,Z 92.580,A 135.574,B 90.000,C 0.000} C_DIS
LIN {X 207.135,Y -202.966,Z 92.702,A 135.582,B 90.000,C 0.000} C_DIS
LIN {X 207.150,Y -202.951,Z 92.792,A 135.587,B 90.000,C 0.000} C_DIS
LIN {X 207.221,Y -202.878,Z 92.868,A 135.607,B 90.000,C 0.000} C_DIS
LIN {X 207.236,Y -202.863,Z 92.959,A 135.611,B 90.000,C 0.000} C_DIS
LIN {X 207.266,Y -202.832,Z 93.080,A 135.619,B 90.000,C 0.000} C_DIS
LIN {X 207.410,Y -202.685,Z 93.323,A 135.660,B 90.000,C 0.000} C_DIS
LIN {X 207.453,Y -202.641,Z 93.638,A 135.672,B 90.000,C 0.000} C_DIS
LIN {X 207.524,Y -202.568,Z 93.761,A 135.692,B 90.000,C 0.000} C_DIS
LIN {X 207.554,Y -202.537,Z 94.067,A 135.701,B 90.000,C 0.000} C_DIS
LIN {X 207.625,Y -202.464,Z 94.195,A 135.721,B 90.000,C 0.000} C_DIS
LIN {X 207.655,Y -202.434,Z 94.501,A 135.729,B 90.000,C 0.000} C_DIS
LIN {X 207.690,Y -202.397,Z 94.565,A 135.739,B 90.000,C 0.000} C_DIS
LIN {X 207.727,Y -202.360,Z 94.727,A 135.750,B 90.000,C 0.000} C_DIS
LIN {X 207.755,Y -202.331,Z 95.558,A 135.758,B 90.000,C 0.000} C_DIS
LIN {X 207.791,Y -202.294,Z 95.721,A 135.768,B 90.000,C 0.000} C_DIS
LIN {X 207.827,Y -202.257,Z 95.806,A 135.778,B 90.000,C 0.000} C_DIS
LIN {X 207.842,Y -202.242,Z 96.010,A 135.782,B 90.000,C 0.000} C_DIS
LIN {X 207.827,Y -202.257,Z 96.214,A 135.778,B 90.000,C 0.000} C_DIS
LIN {X 207.791,Y -202.294,Z 96.299,A 135.768,B 90.000,C 0.000} C_DIS
LIN {X 207.755,Y -202.331,Z 96.443,A 135.758,B 90.000,C 0.000} C_DIS
LIN {X 207.726,Y -202.360,Z 97.166,A 135.750,B 90.000,C 0.000} C_DIS
LIN {X 207.690,Y -202.397,Z 97.311,A 135.739,B 90.000,C 0.000} C_DIS
LIN {X 207.655,Y -202.434,Z 97.396,A 135.729,B 90.000,C 0.000} C_DIS
LIN {X 207.625,Y -202.464,Z 97.804,A 135.721,B 90.000,C 0.000} C_DIS
LIN {X 207.590,Y -202.501,Z 97.889,A 135.711,B 90.000,C 0.000} C_DIS
LIN {X 207.554,Y -202.537,Z 97.952,A 135.701,B 90.000,C 0.000} C_DIS
LIN {X 207.524,Y -202.568,Z 98.259,A 135.692,B 90.000,C 0.000} C_DIS
LIN {X 207.489,Y -202.604,Z 98.322,A 135.682,B 90.000,C 0.000} C_DIS
LIN {X 207.453,Y -202.641,Z 98.365,A 135.672,B 90.000,C 0.000} C_DIS
LIN {X 207.423,Y -202.671,Z 98.569,A 135.664,B 90.000,C 0.000} C_DIS
LIN {X 207.352,Y -202.744,Z 98.654,A 135.644,B 90.000,C 0.000} C_DIS
LIN {X 207.322,Y -202.774,Z 98.858,A 135.635,B 90.000,C 0.000} C_DIS
LIN {X 207.251,Y -202.847,Z 98.938,A 135.615,B 90.000,C 0.000} C_DIS
LIN {X 207.236,Y -202.863,Z 99.029,A 135.611,B 90.000,C 0.000} C_DIS
LIN {X 207.206,Y -202.893,Z 99.150,A 135.603,B 90.000,C 0.000} C_DIS
LIN {X 207.063,Y -203.039,Z 99.365,A 135.562,B 90.000,C 0.000} C_DIS
LIN {X 206.989,Y -203.115,Z 99.595,A 135.541,B 90.000,C 0.000} C_DIS
LIN {X 206.738,Y -203.370,Z 100.001,A 135.471,B 90.000,C 0.000} C_DIS
LIN {X 206.756,Y -203.352,Z 100.045,A 135.476,B 90.000,C 0.000} C_DIS
LIN {X 206.903,Y -203.203,Z 100.078,A 135.517,B 90.000,C 0.000} C_DIS
LIN {X 206.962,Y -203.142,Z 100.180,A 135.534,B 90.000,C 0.000} C_DIS
LIN {X 207.105,Y -202.996,Z 100.222,A 135.574,B 90.000,C 0.000} C_DIS
LIN {X 207.135,Y -202.966,Z 100.273,A 135.582,B 90.000,C 0.000} C_DIS
LIN {X 207.179,Y -202.920,Z 100.324,A 135.595,B 90.000,C 0.000} C_DIS
LIN {X 207.394,Y -202.701,Z 100.367,A 135.656,B 90.000,C 0.000} C_DIS
LIN {X 207.483,Y -202.610,Z 100.469,A 135.681,B 90.000,C 0.000} C_DIS
LIN {X 207.696,Y -202.391,Z 100.511,A 135.741,B 90.000,C 0.000} C_DIS
LIN {X 207.785,Y -202.300,Z 100.614,A 135.766,B 90.000,C 0.000} C_DIS
LIN {X 207.999,Y -202.080,Z 100.656,A 135.827,B 90.000,C 0.000} C_DIS
LIN {X 208.043,Y -202.035,Z 100.707,A 135.839,B 90.000,C 0.000} C_DIS
LIN {X 208.073,Y -202.004,Z 100.758,A 135.848,B 90.000,C 0.000} C_DIS
LIN {X 208.215,Y -201.858,Z 100.801,A 135.888,B 90.000,C 0.000} C_DIS
LIN {X 208.244,Y -201.827,Z 100.852,A 135.897,B 90.000,C 0.000} C_DIS
LIN {X 208.289,Y -201.782,Z 100.903,A 135.909,B 90.000,C 0.000} C_DIS
LIN {X 208.502,Y -201.561,Z 100.945,A 135.970,B 90.000,C 0.000} C_DIS
LIN {X 208.590,Y -201.470,Z 101.047,A 135.995,B 90.000,C 0.000} C_DIS
LIN {X 208.803,Y -201.250,Z 101.090,A 136.055,B 90.000,C 0.000} C_DIS
LIN {X 208.847,Y -201.204,Z 101.141,A 136.068,B 90.000,C 0.000} C_DIS
LIN {X 208.876,Y -201.173,Z 101.192,A 136.076,B 90.000,C 0.000} C_DIS
LIN {X 209.018,Y -201.026,Z 101.234,A 136.117,B 90.000,C 0.000} C_DIS
LIN {X 209.047,Y -200.995,Z 101.285,A 136.125,B 90.000,C 0.000} C_DIS
LIN {X 209.092,Y -200.949,Z 101.336,A 136.138,B 90.000,C 0.000} C_DIS
LIN {X 209.304,Y -200.729,Z 101.379,A 136.198,B 90.000,C 0.000} C_DIS
LIN {X 209.392,Y -200.637,Z 101.481,A 136.223,B 90.000,C 0.000} C_DIS
LIN {X 209.604,Y -200.415,Z 101.523,A 136.284,B 90.000,C 0.000} C_DIS
LIN {X 209.692,Y -200.323,Z 101.625,A 136.309,B 90.000,C 0.000} C_DIS
LIN {X 209.903,Y -200.102,Z 101.668,A 136.369,B 90.000,C 0.000} C_DIS
LIN {X 209.947,Y -200.056,Z 101.719,A 136.382,B 90.000,C 0.000} C_DIS
LIN {X 209.976,Y -200.025,Z 101.770,A 136.390,B 90.000,C 0.000} C_DIS
LIN {X 210.117,Y -199.877,Z 101.812,A 136.431,B 90.000,C 0.000} C_DIS
LIN {X 210.146,Y -199.846,Z 101.863,A 136.439,B 90.000,C 0.000} C_DIS
LIN {X 210.190,Y -199.800,Z 101.914,A 136.452,B 90.000,C 0.000} C_DIS
LIN {X 210.401,Y -199.578,Z 101.957,A 136.512,B 90.000,C 0.000} C_DIS
LIN {X 210.489,Y -199.486,Z 102.059,A 136.537,B 90.000,C 0.000} C_DIS
LIN {X 210.699,Y -199.263,Z 102.101,A 136.598,B 90.000,C 0.000} C_DIS
LIN {X 210.787,Y -199.171,Z 102.203,A 136.623,B 90.000,C 0.000} C_DIS
LIN {X 210.997,Y -198.948,Z 102.246,A 136.683,B 90.000,C 0.000} C_DIS
LIN {X 211.040,Y -198.902,Z 102.297,A 136.696,B 90.000,C 0.000} C_DIS
LIN {X 211.070,Y -198.871,Z 102.348,A 136.704,B 90.000,C 0.000} C_DIS
LIN {X 211.210,Y -198.722,Z 102.390,A 136.745,B 90.000,C 0.000} C_DIS
LIN {X 211.239,Y -198.691,Z 102.441,A 136.753,B 90.000,C 0.000} C_DIS
LIN {X 211.282,Y -198.645,Z 102.492,A 136.766,B 90.000,C 0.000} C_DIS
LIN {X 211.492,Y -198.422,Z 102.535,A 136.826,B 90.000,C 0.000} C_DIS
LIN {X 211.579,Y -198.329,Z 102.637,A 136.851,B 90.000,C 0.000} C_DIS
LIN {X 211.788,Y -198.105,Z 102.679,A 136.912,B 90.000,C 0.000} C_DIS
LIN {X 211.875,Y -198.012,Z 102.781,A 136.937,B 90.000,C 0.000} C_DIS
LIN {X 212.084,Y -197.788,Z 102.824,A 136.998,B 90.000,C 0.000} C_DIS
LIN {X 212.128,Y -197.742,Z 102.875,A 137.010,B 90.000,C 0.000} C_DIS
LIN {X 212.157,Y -197.711,Z 102.926,A 137.019,B 90.000,C 0.000} C_DIS
LIN {X 212.296,Y -197.561,Z 102.968,A 137.059,B 90.000,C 0.000} C_DIS
LIN {X 212.325,Y -197.530,Z 103.019,A 137.067,B 90.000,C 0.000} C_DIS
LIN {X 212.368,Y -197.484,Z 103.070,A 137.080,B 90.000,C 0.000} C_DIS
LIN {X 212.576,Y -197.259,Z 103.113,A 137.140,B 90.000,C 0.000} C_DIS
LIN {X 212.663,Y -197.166,Z 103.215,A 137.166,B 90.000,C 0.000} C_DIS
LIN {X 212.871,Y -196.941,Z 103.257,A 137.226,B 90.000,C 0.000} C_DIS
LIN {X 212.958,Y -196.848,Z 103.360,A 137.251,B 90.000,C 0.000} C_DIS
LIN {X 213.165,Y -196.623,Z 103.402,A 137.312,B 90.000,C 0.000} C_DIS
LIN {X 213.209,Y -196.576,Z 103.453,A 137.324,B 90.000,C 0.000} C_DIS
LIN {X 213.237,Y -196.545,Z 103.504,A 137.333,B 90.000,C 0.000} C_DIS
LIN {X 213.376,Y -196.395,Z 103.547,A 137.373,B 90.000,C 0.000} C_DIS
LIN {X 213.404,Y -196.363,Z 103.598,A 137.381,B 90.000,C 0.000} C_DIS
LIN {X 213.447,Y -196.317,Z 103.649,A 137.394,B 90.000,C 0.000} C_DIS
LIN {X 213.655,Y -196.091,Z 103.691,A 137.454,B 90.000,C 0.000} C_DIS
LIN {X 213.741,Y -195.997,Z 103.793,A 137.480,B 90.000,C 0.000} C_DIS
LIN {X 213.948,Y -195.771,Z 103.836,A 137.540,B 90.000,C 0.000} C_DIS
LIN {X 213.991,Y -195.724,Z 103.887,A 137.553,B 90.000,C 0.000} C_DIS
LIN {X 214.019,Y -195.693,Z 103.938,A 137.561,B 90.000,C 0.000} C_DIS
LIN {X 214.157,Y -195.542,Z 103.980,A 137.601,B 90.000,C 0.000} C_DIS
LIN {X 214.186,Y -195.511,Z 104.031,A 137.610,B 90.000,C 0.000} C_DIS
LIN {X 214.229,Y -195.464,Z 104.082,A 137.622,B 90.000,C 0.000} C_DIS
LIN {X 214.435,Y -195.238,Z 104.125,A 137.683,B 90.000,C 0.000} C_DIS
LIN {X 214.521,Y -195.143,Z 104.227,A 137.708,B 90.000,C 0.000} C_DIS
LIN {X 214.726,Y -194.917,Z 104.269,A 137.769,B 90.000,C 0.000} C_DIS
LIN {X 214.812,Y -194.822,Z 104.371,A 137.794,B 90.000,C 0.000} C_DIS
LIN {X 215.018,Y -194.596,Z 104.414,A 137.854,B 90.000,C 0.000} C_DIS
LIN {X 215.060,Y -194.548,Z 104.465,A 137.867,B 90.000,C 0.000} C_DIS
LIN {X 215.089,Y -194.517,Z 104.516,A 137.875,B 90.000,C 0.000} C_DIS
LIN {X 215.226,Y -194.365,Z 104.558,A 137.916,B 90.000,C 0.000} C_DIS
LIN {X 215.254,Y -194.334,Z 104.609,A 137.924,B 90.000,C 0.000} C_DIS
LIN {X 215.297,Y -194.287,Z 104.660,A 137.937,B 90.000,C 0.000} C_DIS
LIN {X 215.502,Y -194.059,Z 104.703,A 137.997,B 90.000,C 0.000} C_DIS
LIN {X 215.587,Y -193.964,Z 104.805,A 138.022,B 90.000,C 0.000} C_DIS
LIN {X 215.792,Y -193.737,Z 104.847,A 138.083,B 90.000,C 0.000} C_DIS
LIN {X 215.877,Y -193.642,Z 104.949,A 138.108,B 90.000,C 0.000} C_DIS
LIN {X 216.081,Y -193.414,Z 104.992,A 138.168,B 90.000,C 0.000} C_DIS
LIN {X 216.124,Y -193.366,Z 105.043,A 138.181,B 90.000,C 0.000} C_DIS
LIN {X 216.152,Y -193.335,Z 105.094,A 138.189,B 90.000,C 0.000} C_DIS
LIN {X 216.288,Y -193.183,Z 105.136,A 138.230,B 90.000,C 0.000} C_DIS
LIN {X 216.316,Y -193.151,Z 105.187,A 138.238,B 90.000,C 0.000} C_DIS
LIN {X 216.359,Y -193.103,Z 105.238,A 138.251,B 90.000,C 0.000} C_DIS
LIN {X 216.562,Y -192.875,Z 105.281,A 138.311,B 90.000,C 0.000} C_DIS
LIN {X 216.647,Y -192.780,Z 105.383,A 138.336,B 90.000,C 0.000} C_DIS
LIN {X 216.851,Y -192.551,Z 105.425,A 138.397,B 90.000,C 0.000} C_DIS
LIN {X 216.893,Y -192.503,Z 105.476,A 138.409,B 90.000,C 0.000} C_DIS
LIN {X 216.921,Y -192.471,Z 105.527,A 138.418,B 90.000,C 0.000} C_DIS
LIN {X 217.056,Y -192.319,Z 105.570,A 138.458,B 90.000,C 0.000} C_DIS
LIN {X 217.085,Y -192.287,Z 105.621,A 138.466,B 90.000,C 0.000} C_DIS
LIN {X 217.127,Y -192.239,Z 105.672,A 138.479,B 90.000,C 0.000} C_DIS
LIN {X 217.330,Y -192.010,Z 105.714,A 138.540,B 90.000,C 0.000} C_DIS
LIN {X 217.414,Y -191.914,Z 105.817,A 138.565,B 90.000,C 0.000} C_DIS
LIN {X 217.617,Y -191.685,Z 105.859,A 138.625,B 90.000,C 0.000} C_DIS
LIN {X 217.701,Y -191.589,Z 105.961,A 138.650,B 90.000,C 0.000} C_DIS
LIN {X 217.903,Y -191.359,Z 106.004,A 138.711,B 90.000,C 0.000} C_DIS
LIN {X 217.945,Y -191.311,Z 106.055,A 138.723,B 90.000,C 0.000} C_DIS
LIN {X 217.973,Y -191.279,Z 106.106,A 138.732,B 90.000,C 0.000} C_DIS
LIN {X 218.108,Y -191.126,Z 106.148,A 138.772,B 90.000,C 0.000} C_DIS
LIN {X 218.136,Y -191.094,Z 106.199,A 138.781,B 90.000,C 0.000} C_DIS
LIN {X 218.177,Y -191.046,Z 106.250,A 138.793,B 90.000,C 0.000} C_DIS
LIN {X 218.379,Y -190.816,Z 106.293,A 138.854,B 90.000,C 0.000} C_DIS
LIN {X 218.463,Y -190.720,Z 106.395,A 138.879,B 90.000,C 0.000} C_DIS
LIN {X 218.664,Y -190.489,Z 106.437,A 138.939,B 90.000,C 0.000} C_DIS
LIN {X 218.748,Y -190.393,Z 106.539,A 138.964,B 90.000,C 0.000} C_DIS
LIN {X 218.949,Y -190.162,Z 106.582,A 139.025,B 90.000,C 0.000} C_DIS
LIN {X 218.990,Y -190.114,Z 106.633,A 139.038,B 90.000,C 0.000} C_DIS
LIN {X 219.018,Y -190.082,Z 106.684,A 139.046,B 90.000,C 0.000} C_DIS
LIN {X 219.152,Y -189.927,Z 106.726,A 139.086,B 90.000,C 0.000} C_DIS
LIN {X 219.180,Y -189.895,Z 106.777,A 139.095,B 90.000,C 0.000} C_DIS
LIN {X 219.222,Y -189.847,Z 106.828,A 139.107,B 90.000,C 0.000} C_DIS
LIN {X 219.422,Y -189.616,Z 106.871,A 139.168,B 90.000,C 0.000} C_DIS
LIN {X 219.505,Y -189.519,Z 106.973,A 139.193,B 90.000,C 0.000} C_DIS
LIN {X 219.705,Y -189.287,Z 107.015,A 139.253,B 90.000,C 0.000} C_DIS
LIN {X 219.747,Y -189.239,Z 107.066,A 139.266,B 90.000,C 0.000} C_DIS
LIN {X 219.774,Y -189.207,Z 107.117,A 139.274,B 90.000,C 0.000} C_DIS
LIN {X 219.908,Y -189.052,Z 107.160,A 139.315,B 90.000,C 0.000} C_DIS
LIN {X 219.935,Y -189.020,Z 107.211,A 139.323,B 90.000,C 0.000} C_DIS
LIN {X 219.977,Y -188.972,Z 107.262,A 139.336,B 90.000,C 0.000} C_DIS
LIN {X 220.176,Y -188.739,Z 107.304,A 139.396,B 90.000,C 0.000} C_DIS
LIN {X 220.259,Y -188.642,Z 107.406,A 139.421,B 90.000,C 0.000} C_DIS
LIN {X 220.458,Y -188.410,Z 107.449,A 139.482,B 90.000,C 0.000} C_DIS
LIN {X 220.541,Y -188.313,Z 107.551,A 139.507,B 90.000,C 0.000} C_DIS
LIN {X 220.740,Y -188.080,Z 107.593,A 139.568,B 90.000,C 0.000} C_DIS
LIN {X 220.781,Y -188.031,Z 107.644,A 139.580,B 90.000,C 0.000} C_DIS
LIN {X 220.808,Y -187.999,Z 107.695,A 139.588,B 90.000,C 0.000} C_DIS
LIN {X 220.941,Y -187.844,Z 107.738,A 139.629,B 90.000,C 0.000} C_DIS
LIN {X 220.968,Y -187.811,Z 107.789,A 139.637,B 90.000,C 0.000} C_DIS
LIN {X 221.009,Y -187.763,Z 107.840,A 139.650,B 90.000,C 0.000} C_DIS
LIN {X 221.207,Y -187.529,Z 107.882,A 139.710,B 90.000,C 0.000} C_DIS
LIN {X 221.290,Y -187.432,Z 107.984,A 139.735,B 90.000,C 0.000} C_DIS
LIN {X 221.488,Y -187.198,Z 108.027,A 139.796,B 90.000,C 0.000} C_DIS
LIN {X 221.570,Y -187.101,Z 108.129,A 139.821,B 90.000,C 0.000} C_DIS
LIN {X 221.767,Y -186.867,Z 108.171,A 139.882,B 90.000,C 0.000} C_DIS
LIN {X 221.808,Y -186.818,Z 108.222,A 139.894,B 90.000,C 0.000} C_DIS
LIN {X 221.836,Y -186.786,Z 108.274,A 139.903,B 90.000,C 0.000} C_DIS
LIN {X 221.967,Y -186.630,Z 108.316,A 139.943,B 90.000,C 0.000} C_DIS
LIN {X 221.994,Y -186.597,Z 108.367,A 139.951,B 90.000,C 0.000} C_DIS
LIN {X 222.035,Y -186.548,Z 108.418,A 139.964,B 90.000,C 0.000} C_DIS
LIN {X 222.232,Y -186.314,Z 108.460,A 140.024,B 90.000,C 0.000} C_DIS
LIN {X 222.314,Y -186.216,Z 108.563,A 140.050,B 90.000,C 0.000} C_DIS
LIN {X 222.511,Y -185.981,Z 108.605,A 140.110,B 90.000,C 0.000} C_DIS
LIN {X 222.592,Y -185.884,Z 108.707,A 140.135,B 90.000,C 0.000} C_DIS
LIN {X 222.788,Y -185.648,Z 108.750,A 140.196,B 90.000,C 0.000} C_DIS
LIN {X 222.829,Y -185.600,Z 108.801,A 140.208,B 90.000,C 0.000} C_DIS
LIN {X 222.856,Y -185.567,Z 108.852,A 140.217,B 90.000,C 0.000} C_DIS
LIN {X 222.987,Y -185.410,Z 108.894,A 140.257,B 90.000,C 0.000} C_DIS
LIN {X 223.014,Y -185.377,Z 108.945,A 140.265,B 90.000,C 0.000} C_DIS
LIN {X 223.055,Y -185.328,Z 108.996,A 140.278,B 90.000,C 0.000} C_DIS
LIN {X 223.250,Y -185.093,Z 109.039,A 140.338,B 90.000,C 0.000} C_DIS
LIN {X 223.332,Y -184.995,Z 109.141,A 140.364,B 90.000,C 0.000} C_DIS
LIN {X 223.527,Y -184.759,Z 109.183,A 140.424,B 90.000,C 0.000} C_DIS
LIN {X 223.608,Y -184.661,Z 109.285,A 140.449,B 90.000,C 0.000} C_DIS
LIN {X 223.803,Y -184.424,Z 109.328,A 140.510,B 90.000,C 0.000} C_DIS
LIN {X 223.843,Y -184.375,Z 109.379,A 140.522,B 90.000,C 0.000} C_DIS
LIN {X 223.870,Y -184.342,Z 109.430,A 140.531,B 90.000,C 0.000} C_DIS
LIN {X 224.000,Y -184.185,Z 109.472,A 140.571,B 90.000,C 0.000} C_DIS
LIN {X 224.027,Y -184.152,Z 109.523,A 140.580,B 90.000,C 0.000} C_DIS
LIN {X 224.067,Y -184.103,Z 109.574,A 140.592,B 90.000,C 0.000} C_DIS
LIN {X 224.262,Y -183.866,Z 109.617,A 140.653,B 90.000,C 0.000} C_DIS
LIN {X 224.342,Y -183.768,Z 109.719,A 140.678,B 90.000,C 0.000} C_DIS
LIN {X 224.536,Y -183.531,Z 109.761,A 140.738,B 90.000,C 0.000} C_DIS
LIN {X 224.577,Y -183.481,Z 109.812,A 140.751,B 90.000,C 0.000} C_DIS
LIN {X 224.603,Y -183.448,Z 109.863,A 140.759,B 90.000,C 0.000} C_DIS
LIN {X 224.732,Y -183.290,Z 109.906,A 140.800,B 90.000,C 0.000} C_DIS
LIN {X 224.759,Y -183.257,Z 109.957,A 140.808,B 90.000,C 0.000} C_DIS
LIN {X 224.800,Y -183.208,Z 110.008,A 140.821,B 90.000,C 0.000} C_DIS
LIN {X 224.993,Y -182.970,Z 110.050,A 140.881,B 90.000,C 0.000} C_DIS
LIN {X 225.073,Y -182.872,Z 110.152,A 140.906,B 90.000,C 0.000} C_DIS
LIN {X 225.266,Y -182.634,Z 110.195,A 140.967,B 90.000,C 0.000} C_DIS
LIN {X 225.346,Y -182.535,Z 110.297,A 140.992,B 90.000,C 0.000} C_DIS
LIN {X 225.539,Y -182.297,Z 110.339,A 141.052,B 90.000,C 0.000} C_DIS
LIN {X 225.579,Y -182.247,Z 110.390,A 141.065,B 90.000,C 0.000} C_DIS
LIN {X 225.606,Y -182.214,Z 110.441,A 141.073,B 90.000,C 0.000} C_DIS
LIN {X 225.734,Y -182.055,Z 110.484,A 141.114,B 90.000,C 0.000} C_DIS
LIN {X 225.761,Y -182.022,Z 110.535,A 141.122,B 90.000,C 0.000} C_DIS
LIN {X 225.801,Y -181.973,Z 110.586,A 141.135,B 90.000,C 0.000} C_DIS
LIN {X 225.993,Y -181.734,Z 110.628,A 141.195,B 90.000,C 0.000} C_DIS
LIN {X 226.072,Y -181.635,Z 110.730,A 141.220,B 90.000,C 0.000} C_DIS
LIN {X 226.264,Y -181.396,Z 110.773,A 141.281,B 90.000,C 0.000} C_DIS
LIN {X 226.344,Y -181.297,Z 110.875,A 141.306,B 90.000,C 0.000} C_DIS
LIN {X 226.535,Y -181.058,Z 110.917,A 141.366,B 90.000,C 0.000} C_DIS
LIN {X 226.575,Y -181.008,Z 110.969,A 141.379,B 90.000,C 0.000} C_DIS
LIN {X 226.601,Y -180.975,Z 111.020,A 141.387,B 90.000,C 0.000} C_DIS
LIN {X 226.729,Y -180.815,Z 111.062,A 141.428,B 90.000,C 0.000} C_DIS
LIN {X 226.755,Y -180.782,Z 111.113,A 141.436,B 90.000,C 0.000} C_DIS
LIN {X 226.795,Y -180.732,Z 111.164,A 141.449,B 90.000,C 0.000} C_DIS
LIN {X 226.985,Y -180.493,Z 111.207,A 141.509,B 90.000,C 0.000} C_DIS
LIN {X 227.065,Y -180.393,Z 111.309,A 141.534,B 90.000,C 0.000} C_DIS
LIN {X 227.255,Y -180.153,Z 111.351,A 141.595,B 90.000,C 0.000} C_DIS
LIN {X 227.295,Y -180.103,Z 111.402,A 141.607,B 90.000,C 0.000} C_DIS
LIN {X 227.321,Y -180.070,Z 111.453,A 141.616,B 90.000,C 0.000} C_DIS
LIN {X 227.448,Y -179.910,Z 111.496,A 141.656,B 90.000,C 0.000} C_DIS
LIN {X 227.474,Y -179.877,Z 111.547,A 141.665,B 90.000,C 0.000} C_DIS
LIN {X 227.514,Y -179.827,Z 111.598,A 141.677,B 90.000,C 0.000} C_DIS
LIN {X 227.703,Y -179.586,Z 111.640,A 141.738,B 90.000,C 0.000} C_DIS
LIN {X 227.782,Y -179.486,Z 111.742,A 141.763,B 90.000,C 0.000} C_DIS
LIN {X 227.972,Y -179.246,Z 111.785,A 141.823,B 90.000,C 0.000} C_DIS
LIN {X 228.050,Y -179.145,Z 111.887,A 141.848,B 90.000,C 0.000} C_DIS
LIN {X 228.239,Y -178.905,Z 111.929,A 141.909,B 90.000,C 0.000} C_DIS
LIN {X 228.279,Y -178.854,Z 111.980,A 141.922,B 90.000,C 0.000} C_DIS
LIN {X 228.305,Y -178.821,Z 112.031,A 141.930,B 90.000,C 0.000} C_DIS
LIN {X 228.431,Y -178.660,Z 112.074,A 141.970,B 90.000,C 0.000} C_DIS
LIN {X 228.457,Y -178.627,Z 112.125,A 141.979,B 90.000,C 0.000} C_DIS
LIN {X 228.496,Y -178.577,Z 112.176,A 141.991,B 90.000,C 0.000} C_DIS
LIN {X 228.684,Y -178.335,Z 112.218,A 142.052,B 90.000,C 0.000} C_DIS
LIN {X 228.763,Y -178.235,Z 112.320,A 142.077,B 90.000,C 0.000} C_DIS
LIN {X 228.951,Y -177.993,Z 112.363,A 142.137,B 90.000,C 0.000} C_DIS
LIN {X 229.029,Y -177.893,Z 112.465,A 142.163,B 90.000,C 0.000} C_DIS
LIN {X 229.217,Y -177.651,Z 112.507,A 142.223,B 90.000,C 0.000} C_DIS
LIN {X 229.256,Y -177.600,Z 112.558,A 142.236,B 90.000,C 0.000} C_DIS
LIN {X 229.282,Y -177.567,Z 112.609,A 142.244,B 90.000,C 0.000} C_DIS
LIN {X 229.407,Y -177.405,Z 112.652,A 142.284,B 90.000,C 0.000} C_DIS
LIN {X 229.433,Y -177.372,Z 112.703,A 142.293,B 90.000,C 0.000} C_DIS
LIN {X 229.471,Y -177.321,Z 112.754,A 142.305,B 90.000,C 0.000} C_DIS
LIN {X 229.659,Y -177.079,Z 112.796,A 142.366,B 90.000,C 0.000} C_DIS
LIN {X 229.736,Y -176.978,Z 112.898,A 142.391,B 90.000,C 0.000} C_DIS
LIN {X 229.923,Y -176.735,Z 112.941,A 142.452,B 90.000,C 0.000} C_DIS
LIN {X 230.001,Y -176.634,Z 113.043,A 142.477,B 90.000,C 0.000} C_DIS
LIN {X 230.187,Y -176.391,Z 113.085,A 142.537,B 90.000,C 0.000} C_DIS
LIN {X 230.226,Y -176.341,Z 113.136,A 142.550,B 90.000,C 0.000} C_DIS
LIN {X 230.252,Y -176.307,Z 113.187,A 142.558,B 90.000,C 0.000} C_DIS
LIN {X 230.376,Y -176.145,Z 113.230,A 142.599,B 90.000,C 0.000} C_DIS
LIN {X 230.401,Y -176.111,Z 113.281,A 142.607,B 90.000,C 0.000} C_DIS
LIN {X 230.440,Y -176.061,Z 113.332,A 142.619,B 90.000,C 0.000} C_DIS
LIN {X 230.626,Y -175.817,Z 113.374,A 142.680,B 90.000,C 0.000} C_DIS
LIN {X 230.703,Y -175.716,Z 113.477,A 142.705,B 90.000,C 0.000} C_DIS
LIN {X 230.888,Y -175.472,Z 113.519,A 142.766,B 90.000,C 0.000} C_DIS
LIN {X 230.927,Y -175.422,Z 113.570,A 142.778,B 90.000,C 0.000} C_DIS
LIN {X 230.953,Y -175.388,Z 113.621,A 142.787,B 90.000,C 0.000} C_DIS
LIN {X 231.076,Y -175.225,Z 113.664,A 142.827,B 90.000,C 0.000} C_DIS
LIN {X 231.102,Y -175.191,Z 113.715,A 142.835,B 90.000,C 0.000} C_DIS
LIN {X 231.140,Y -175.141,Z 113.766,A 142.848,B 90.000,C 0.000} C_DIS
LIN {X 231.325,Y -174.896,Z 113.808,A 142.908,B 90.000,C 0.000} C_DIS
LIN {X 231.402,Y -174.795,Z 113.910,A 142.934,B 90.000,C 0.000} C_DIS
LIN {X 231.586,Y -174.550,Z 113.953,A 142.994,B 90.000,C 0.000} C_DIS
LIN {X 231.663,Y -174.449,Z 114.055,A 143.019,B 90.000,C 0.000} C_DIS
LIN {X 231.847,Y -174.204,Z 114.097,A 143.080,B 90.000,C 0.000} C_DIS
LIN {X 231.885,Y -174.153,Z 114.148,A 143.092,B 90.000,C 0.000} C_DIS
LIN {X 231.911,Y -174.119,Z 114.199,A 143.101,B 90.000,C 0.000} C_DIS
LIN {X 232.033,Y -173.956,Z 114.242,A 143.141,B 90.000,C 0.000} C_DIS
LIN {X 232.059,Y -173.922,Z 114.293,A 143.149,B 90.000,C 0.000} C_DIS
LIN {X 232.097,Y -173.871,Z 114.344,A 143.162,B 90.000,C 0.000} C_DIS
LIN {X 232.280,Y -173.626,Z 114.386,A 143.223,B 90.000,C 0.000} C_DIS
LIN {X 232.357,Y -173.524,Z 114.488,A 143.248,B 90.000,C 0.000} C_DIS
LIN {X 232.540,Y -173.278,Z 114.531,A 143.308,B 90.000,C 0.000} C_DIS
LIN {X 232.615,Y -173.177,Z 114.633,A 143.333,B 90.000,C 0.000} C_DIS
LIN {X 232.798,Y -172.931,Z 114.680,A 143.394,B 90.000,C 0.000} C_DIS
LIN {X 232.847,Y -172.865,Z 114.744,A 143.410,B 90.000,C 0.000} C_DIS
LIN {X 232.881,Y -172.819,Z 114.770,A 143.421,B 90.000,C 0.000} C_DIS
LIN {X 232.936,Y -172.745,Z 114.717,A 143.439,B 90.000,C 0.000} C_DIS
LIN {X 232.986,Y -172.677,Z 114.620,A 143.456,B 90.000,C 0.000} C_DIS
LIN {X 233.009,Y -172.647,Z 114.513,A 143.464,B 90.000,C 0.000} C_DIS
LIN {X 233.069,Y -172.566,Z 114.348,A 143.483,B 90.000,C 0.000} C_DIS
LIN {X 233.357,Y -172.176,Z 113.883,A 143.579,B 90.000,C 0.000} C_DIS
LIN {X 233.458,Y -172.038,Z 113.787,A 143.613,B 90.000,C 0.000} C_DIS
LIN {X 233.505,Y -171.976,Z 113.766,A 143.628,B 90.000,C 0.000} C_DIS
LIN {X 233.524,Y -171.949,Z 113.715,A 143.635,B 90.000,C 0.000} C_DIS
LIN {X 233.717,Y -171.687,Z 113.661,A 143.699,B 90.000,C 0.000} C_DIS
LIN {X 234.782,Y -170.228,Z 113.661,A 144.056,B 90.000,C 0.000} C_DIS
LIN {X 235.152,Y -169.716,Z 113.768,A 144.181,B 90.000,C 0.000} C_DIS
LIN {X 236.142,Y -168.336,Z 113.806,A 144.516,B 90.000,C 0.000} C_DIS
LIN {X 236.488,Y -167.850,Z 113.912,A 144.634,B 90.000,C 0.000} C_DIS
LIN {X 237.404,Y -166.551,Z 113.951,A 144.948,B 90.000,C 0.000} C_DIS
LIN {X 237.746,Y -166.063,Z 114.057,A 145.066,B 90.000,C 0.000} C_DIS
LIN {X 238.714,Y -164.668,Z 114.095,A 145.402,B 90.000,C 0.000} C_DIS
LIN {X 239.052,Y -164.177,Z 114.201,A 145.519,B 90.000,C 0.000} C_DIS
LIN {X 239.949,Y -162.864,Z 114.240,A 145.834,B 90.000,C 0.000} C_DIS
LIN {X 240.288,Y -162.362,Z 114.346,A 145.953,B 90.000,C 0.000} C_DIS
LIN {X 241.443,Y -160.641,Z 114.365,A 146.363,B 90.000,C 0.000} C_DIS
LIN {X 242.440,Y -159.132,Z 112.640,A 146.720,B 90.000,C 0.000} C_DIS
LIN {X 242.555,Y -158.956,Z 112.486,A 146.762,B 90.000,C 0.000} C_DIS
LIN {X 242.614,Y -158.867,Z 112.384,A 146.783,B 90.000,C 0.000} C_DIS
LIN {X 242.734,Y -158.682,Z 112.299,A 146.826,B 90.000,C 0.000} C_DIS
LIN {X 242.853,Y -158.500,Z 112.095,A 146.869,B 90.000,C 0.000} C_DIS
LIN {X 242.920,Y -158.398,Z 112.052,A 146.893,B 90.000,C 0.000} C_DIS
LIN {X 242.969,Y -158.322,Z 112.031,A 146.911,B 90.000,C 0.000} C_DIS
LIN {X 243.011,Y -158.259,Z 111.929,A 146.926,B 90.000,C 0.000} C_DIS
LIN {X 243.060,Y -158.183,Z 111.908,A 146.944,B 90.000,C 0.000} C_DIS
LIN {X 243.126,Y -158.081,Z 111.865,A 146.968,B 90.000,C 0.000} C_DIS
LIN {X 243.258,Y -157.878,Z 111.659,A 147.016,B 90.000,C 0.000} C_DIS
LIN {X 243.430,Y -157.613,Z 111.598,A 147.078,B 90.000,C 0.000} C_DIS
LIN {X 243.462,Y -157.563,Z 111.547,A 147.090,B 90.000,C 0.000} C_DIS
LIN {X 243.485,Y -157.528,Z 111.496,A 147.098,B 90.000,C 0.000} C_DIS
LIN {X 243.596,Y -157.356,Z 111.453,A 147.139,B 90.000,C 0.000} C_DIS
LIN {X 243.642,Y -157.285,Z 111.351,A 147.155,B 90.000,C 0.000} C_DIS
LIN {X 243.753,Y -157.113,Z 111.309,A 147.196,B 90.000,C 0.000} C_DIS
LIN {X 243.776,Y -157.078,Z 111.258,A 147.204,B 90.000,C 0.000} C_DIS
LIN {X 243.810,Y -157.024,Z 111.207,A 147.217,B 90.000,C 0.000} C_DIS
LIN {X 243.976,Y -156.767,Z 111.164,A 147.277,B 90.000,C 0.000} C_DIS
LIN {X 244.045,Y -156.659,Z 111.062,A 147.302,B 90.000,C 0.000} C_DIS
LIN {X 244.210,Y -156.402,Z 111.020,A 147.363,B 90.000,C 0.000} C_DIS
LIN {X 244.244,Y -156.348,Z 110.969,A 147.376,B 90.000,C 0.000} C_DIS
LIN {X 244.290,Y -156.276,Z 110.917,A 147.392,B 90.000,C 0.000} C_DIS
LIN {X 244.510,Y -155.932,Z 110.875,A 147.473,B 90.000,C 0.000} C_DIS
LIN {X 244.556,Y -155.861,Z 110.824,A 147.490,B 90.000,C 0.000} C_DIS
LIN {X 244.624,Y -155.754,Z 110.773,A 147.515,B 90.000,C 0.000} C_DIS
LIN {X 244.953,Y -155.236,Z 110.731,A 147.636,B 90.000,C 0.000} C_DIS
LIN {X 245.021,Y -155.129,Z 110.679,A 147.661,B 90.000,C 0.000} C_DIS
LIN {X 245.223,Y -154.808,Z 110.626,A 147.736,B 90.000,C 0.000} C_DIS
LIN {X 246.355,Y -153.001,Z 110.626,A 148.157,B 90.000,C 0.000} C_DIS
LIN {X 246.555,Y -152.679,Z 110.679,A 148.232,B 90.000,C 0.000} C_DIS
LIN {X 246.610,Y -152.589,Z 110.730,A 148.253,B 90.000,C 0.000} C_DIS
LIN {X 246.879,Y -152.154,Z 110.773,A 148.354,B 90.000,C 0.000} C_DIS
LIN {X 246.979,Y -151.992,Z 110.875,A 148.392,B 90.000,C 0.000} C_DIS
LIN {X 247.193,Y -151.644,Z 110.917,A 148.472,B 90.000,C 0.000} C_DIS
LIN {X 247.237,Y -151.571,Z 110.969,A 148.489,B 90.000,C 0.000} C_DIS
LIN {X 247.270,Y -151.517,Z 111.020,A 148.502,B 90.000,C 0.000} C_DIS
LIN {X 247.430,Y -151.256,Z 111.062,A 148.562,B 90.000,C 0.000} C_DIS
LIN {X 247.496,Y -151.147,Z 111.164,A 148.587,B 90.000,C 0.000} C_DIS
LIN {X 247.656,Y -150.886,Z 111.207,A 148.648,B 90.000,C 0.000} C_DIS
LIN {X 247.689,Y -150.831,Z 111.258,A 148.660,B 90.000,C 0.000} C_DIS
LIN {X 247.711,Y -150.795,Z 111.309,A 148.669,B 90.000,C 0.000} C_DIS
LIN {X 247.817,Y -150.621,Z 111.351,A 148.709,B 90.000,C 0.000} C_DIS
LIN {X 247.861,Y -150.548,Z 111.453,A 148.726,B 90.000,C 0.000} C_DIS
LIN {X 247.967,Y -150.374,Z 111.496,A 148.766,B 90.000,C 0.000} C_DIS
LIN {X 247.989,Y -150.337,Z 111.547,A 148.775,B 90.000,C 0.000} C_DIS
LIN {X 248.020,Y -150.287,Z 111.598,A 148.786,B 90.000,C 0.000} C_DIS
LIN {X 248.183,Y -150.017,Z 111.659,A 148.849,B 90.000,C 0.000} C_DIS
LIN {X 248.309,Y -149.809,Z 111.865,A 148.897,B 90.000,C 0.000} C_DIS
LIN {X 248.371,Y -149.705,Z 111.908,A 148.921,B 90.000,C 0.000} C_DIS
LIN {X 248.418,Y -149.628,Z 111.929,A 148.939,B 90.000,C 0.000} C_DIS
LIN {X 248.457,Y -149.563,Z 112.031,A 148.953,B 90.000,C 0.000} C_DIS
LIN {X 248.504,Y -149.485,Z 112.052,A 148.971,B 90.000,C 0.000} C_DIS
LIN {X 248.567,Y -149.381,Z 112.095,A 148.995,B 90.000,C 0.000} C_DIS
LIN {X 248.677,Y -149.197,Z 112.299,A 149.038,B 90.000,C 0.000} C_DIS
LIN {X 248.795,Y -148.999,Z 112.405,A 149.083,B 90.000,C 0.000} C_DIS
LIN {X 249.736,Y -147.418,Z 114.098,A 149.447,B 90.000,C 0.000} C_DIS
LIN {X 250.104,Y -146.793,Z 114.975,A 149.590,B 90.000,C 0.000} C_DIS
LIN {X 250.136,Y -146.738,Z 115.117,A 149.603,B 90.000,C 0.000} C_DIS
LIN {X 250.147,Y -146.719,Z 115.198,A 149.607,B 90.000,C 0.000} C_DIS
LIN {X 250.198,Y -146.631,Z 115.270,A 149.627,B 90.000,C 0.000} C_DIS
LIN {X 250.209,Y -146.613,Z 115.361,A 149.631,B 90.000,C 0.000} C_DIS
LIN {X 250.231,Y -146.576,Z 115.482,A 149.640,B 90.000,C 0.000} C_DIS
LIN {X 250.334,Y -146.400,Z 115.705,A 149.680,B 90.000,C 0.000} C_DIS
LIN {X 250.355,Y -146.364,Z 115.826,A 149.688,B 90.000,C 0.000} C_DIS
LIN {X 250.366,Y -146.345,Z 115.917,A 149.693,B 90.000,C 0.000} C_DIS
LIN {X 250.417,Y -146.257,Z 115.997,A 149.713,B 90.000,C 0.000} C_DIS
LIN {X 250.439,Y -146.220,Z 116.201,A 149.721,B 90.000,C 0.000} C_DIS
LIN {X 250.490,Y -146.132,Z 116.286,A 149.741,B 90.000,C 0.000} C_DIS
LIN {X 250.512,Y -146.096,Z 116.490,A 149.750,B 90.000,C 0.000} C_DIS
LIN {X 250.537,Y -146.051,Z 116.533,A 149.760,B 90.000,C 0.000} C_DIS
LIN {X 250.563,Y -146.007,Z 116.597,A 149.770,B 90.000,C 0.000} C_DIS
LIN {X 250.584,Y -145.971,Z 116.903,A 149.778,B 90.000,C 0.000} C_DIS
LIN {X 250.610,Y -145.927,Z 116.966,A 149.788,B 90.000,C 0.000} C_DIS
LIN {X 250.636,Y -145.883,Z 117.009,A 149.798,B 90.000,C 0.000} C_DIS
LIN {X 250.657,Y -145.846,Z 117.213,A 149.807,B 90.000,C 0.000} C_DIS
LIN {X 250.683,Y -145.802,Z 117.255,A 149.817,B 90.000,C 0.000} C_DIS
LIN {X 250.708,Y -145.758,Z 117.319,A 149.827,B 90.000,C 0.000} C_DIS
LIN {X 250.730,Y -145.721,Z 117.625,A 149.835,B 90.000,C 0.000} C_DIS
LIN {X 250.755,Y -145.677,Z 117.689,A 149.845,B 90.000,C 0.000} C_DIS
LIN {X 250.781,Y -145.633,Z 117.774,A 149.856,B 90.000,C 0.000} C_DIS
LIN {X 250.802,Y -145.596,Z 118.182,A 149.864,B 90.000,C 0.000} C_DIS
LIN {X 250.854,Y -145.508,Z 118.373,A 149.884,B 90.000,C 0.000} C_DIS
LIN {X 250.875,Y -145.471,Z 118.884,A 149.893,B 90.000,C 0.000} C_DIS
LIN {X 250.901,Y -145.427,Z 118.990,A 149.903,B 90.000,C 0.000} C_DIS
LIN {X 250.927,Y -145.381,Z 119.189,A 149.913,B 90.000,C 0.000} C_DIS
LIN {X 250.947,Y -145.347,Z 120.236,A 149.921,B 90.000,C 0.000} C_DIS
LIN {X 250.973,Y -145.302,Z 120.435,A 149.931,B 90.000,C 0.000} C_DIS
LIN {X 250.999,Y -145.258,Z 120.520,A 149.941,B 90.000,C 0.000} C_DIS
LIN {X 251.009,Y -145.239,Z 120.724,A 149.945,B 90.000,C 0.000} C_DIS
LIN {X 250.999,Y -145.258,Z 120.928,A 149.941,B 90.000,C 0.000} C_DIS
LIN {X 250.973,Y -145.302,Z 121.013,A 149.931,B 90.000,C 0.000} C_DIS
LIN {X 250.947,Y -145.347,Z 121.212,A 149.921,B 90.000,C 0.000} C_DIS
LIN {X 250.927,Y -145.381,Z 122.260,A 149.913,B 90.000,C 0.000} C_DIS
LIN {X 250.901,Y -145.427,Z 122.458,A 149.903,B 90.000,C 0.000} C_DIS
LIN {X 250.875,Y -145.471,Z 122.565,A 149.893,B 90.000,C 0.000} C_DIS
LIN {X 250.854,Y -145.508,Z 123.075,A 149.884,B 90.000,C 0.000} C_DIS
LIN {X 250.828,Y -145.552,Z 123.181,A 149.874,B 90.000,C 0.000} C_DIS
LIN {X 250.802,Y -145.596,Z 123.245,A 149.864,B 90.000,C 0.000} C_DIS
LIN {X 250.781,Y -145.633,Z 123.551,A 149.856,B 90.000,C 0.000} C_DIS
LIN {X 250.730,Y -145.721,Z 123.678,A 149.835,B 90.000,C 0.000} C_DIS
LIN {X 250.708,Y -145.758,Z 123.985,A 149.827,B 90.000,C 0.000} C_DIS
LIN {X 250.657,Y -145.846,Z 124.112,A 149.807,B 90.000,C 0.000} C_DIS
LIN {X 250.636,Y -145.883,Z 124.418,A 149.798,B 90.000,C 0.000} C_DIS
LIN {X 250.610,Y -145.927,Z 124.482,A 149.788,B 90.000,C 0.000} C_DIS
LIN {X 250.584,Y -145.971,Z 124.524,A 149.778,B 90.000,C 0.000} C_DIS
LIN {X 250.563,Y -146.007,Z 124.728,A 149.770,B 90.000,C 0.000} C_DIS
LIN {X 250.512,Y -146.096,Z 124.813,A 149.750,B 90.000,C 0.000} C_DIS
LIN {X 250.490,Y -146.132,Z 125.018,A 149.741,B 90.000,C 0.000} C_DIS
LIN {X 250.439,Y -146.220,Z 125.102,A 149.721,B 90.000,C 0.000} C_DIS
LIN {X 250.417,Y -146.257,Z 125.307,A 149.713,B 90.000,C 0.000} C_DIS
LIN {X 250.366,Y -146.345,Z 125.392,A 149.693,B 90.000,C 0.000} C_DIS
LIN {X 250.344,Y -146.382,Z 125.596,A 149.684,B 90.000,C 0.000} C_DIS
LIN {X 250.293,Y -146.470,Z 125.673,A 149.664,B 90.000,C 0.000} C_DIS
LIN {X 250.260,Y -146.527,Z 125.878,A 149.651,B 90.000,C 0.000} C_DIS
LIN {X 250.150,Y -146.714,Z 126.135,A 149.608,B 90.000,C 0.000} C_DIS
LIN {X 250.184,Y -146.655,Z 126.250,A 149.622,B 90.000,C 0.000} C_DIS
LIN {X 250.252,Y -146.541,Z 126.328,A 149.648,B 90.000,C 0.000} C_DIS
LIN {X 250.401,Y -146.286,Z 126.382,A 149.706,B 90.000,C 0.000} C_DIS
LIN {X 250.460,Y -146.184,Z 126.484,A 149.730,B 90.000,C 0.000} C_DIS
LIN {X 250.614,Y -145.919,Z 126.527,A 149.790,B 90.000,C 0.000} C_DIS
LIN {X 250.678,Y -145.809,Z 126.629,A 149.815,B 90.000,C 0.000} C_DIS
LIN {X 250.832,Y -145.544,Z 126.671,A 149.876,B 90.000,C 0.000} C_DIS
LIN {X 250.864,Y -145.489,Z 126.722,A 149.888,B 90.000,C 0.000} C_DIS
LIN {X 250.886,Y -145.453,Z 126.773,A 149.897,B 90.000,C 0.000} C_DIS
LIN {X 250.988,Y -145.276,Z 126.816,A 149.937,B 90.000,C 0.000} C_DIS
LIN {X 251.009,Y -145.239,Z 126.867,A 149.945,B 90.000,C 0.000} C_DIS
LIN {X 251.041,Y -145.184,Z 126.918,A 149.958,B 90.000,C 0.000} C_DIS
LIN {X 251.194,Y -144.919,Z 126.960,A 150.019,B 90.000,C 0.000} C_DIS
LIN {X 251.258,Y -144.809,Z 127.062,A 150.044,B 90.000,C 0.000} C_DIS
LIN {X 251.411,Y -144.543,Z 127.105,A 150.104,B 90.000,C 0.000} C_DIS
LIN {X 251.442,Y -144.488,Z 127.156,A 150.117,B 90.000,C 0.000} C_DIS
LIN {X 251.463,Y -144.451,Z 127.207,A 150.125,B 90.000,C 0.000} C_DIS
LIN {X 251.565,Y -144.274,Z 127.249,A 150.165,B 90.000,C 0.000} C_DIS
LIN {X 251.586,Y -144.237,Z 127.300,A 150.174,B 90.000,C 0.000} C_DIS
LIN {X 251.617,Y -144.183,Z 127.351,A 150.186,B 90.000,C 0.000} C_DIS
LIN {X 251.769,Y -143.917,Z 127.399,A 150.247,B 90.000,C 0.000} C_DIS
LIN {X 251.836,Y -143.802,Z 127.504,A 150.273,B 90.000,C 0.000} C_DIS
LIN {X 251.885,Y -143.715,Z 127.431,A 150.293,B 90.000,C 0.000} C_DIS
LIN {X 251.931,Y -143.635,Z 127.243,A 150.311,B 90.000,C 0.000} C_DIS
LIN {X 251.955,Y -143.591,Z 126.624,A 150.321,B 90.000,C 0.000} C_DIS
LIN {X 252.006,Y -143.503,Z 126.379,A 150.341,B 90.000,C 0.000} C_DIS
LIN {X 252.027,Y -143.466,Z 125.765,A 150.349,B 90.000,C 0.000} C_DIS
LIN {X 252.077,Y -143.377,Z 125.512,A 150.370,B 90.000,C 0.000} C_DIS
LIN {X 252.098,Y -143.340,Z 124.897,A 150.378,B 90.000,C 0.000} C_DIS
LIN {X 252.149,Y -143.251,Z 124.644,A 150.398,B 90.000,C 0.000} C_DIS
LIN {X 252.170,Y -143.215,Z 124.030,A 150.406,B 90.000,C 0.000} C_DIS
LIN {X 252.220,Y -143.126,Z 123.798,A 150.427,B 90.000,C 0.000} C_DIS
LIN {X 252.241,Y -143.089,Z 123.287,A 150.435,B 90.000,C 0.000} C_DIS
LIN {X 252.291,Y -143.000,Z 123.075,A 150.455,B 90.000,C 0.000} C_DIS
LIN {X 252.312,Y -142.963,Z 122.565,A 150.464,B 90.000,C 0.000} C_DIS
LIN {X 252.338,Y -142.919,Z 122.458,A 150.474,B 90.000,C 0.000} C_DIS
LIN {X 252.363,Y -142.874,Z 122.416,A 150.484,B 90.000,C 0.000} C_DIS
LIN {X 252.373,Y -142.856,Z 122.314,A 150.488,B 90.000,C 0.000} C_DIS
LIN {X 252.391,Y -142.824,Z 122.206,A 150.495,B 90.000,C 0.000} C_DIS
LIN {X 252.444,Y -142.730,Z 122.169,A 150.517,B 90.000,C 0.000} C_DIS
LIN {X 252.495,Y -142.641,Z 122.148,A 150.537,B 90.000,C 0.000} C_DIS
LIN {X 252.515,Y -142.604,Z 122.097,A 150.545,B 90.000,C 0.000} C_DIS
LIN {X 252.547,Y -142.549,Z 122.046,A 150.558,B 90.000,C 0.000} C_DIS
LIN {X 252.697,Y -142.282,Z 122.004,A 150.618,B 90.000,C 0.000} C_DIS
LIN {X 252.760,Y -142.171,Z 121.902,A 150.643,B 90.000,C 0.000} C_DIS
LIN {X 252.910,Y -141.904,Z 121.859,A 150.704,B 90.000,C 0.000} C_DIS
LIN {X 252.941,Y -141.848,Z 121.808,A 150.716,B 90.000,C 0.000} C_DIS
LIN {X 252.982,Y -141.774,Z 121.757,A 150.733,B 90.000,C 0.000} C_DIS
LIN {X 253.182,Y -141.418,Z 121.715,A 150.814,B 90.000,C 0.000} C_DIS
LIN {X 253.264,Y -141.270,Z 121.613,A 150.847,B 90.000,C 0.000} C_DIS
LIN {X 253.463,Y -140.913,Z 121.570,A 150.928,B 90.000,C 0.000} C_DIS
LIN {X 253.504,Y -140.839,Z 121.519,A 150.945,B 90.000,C 0.000} C_DIS
LIN {X 253.535,Y -140.783,Z 121.468,A 150.957,B 90.000,C 0.000} C_DIS
LIN {X 253.684,Y -140.515,Z 121.426,A 151.018,B 90.000,C 0.000} C_DIS
LIN {X 253.715,Y -140.460,Z 121.375,A 151.031,B 90.000,C 0.000} C_DIS
LIN {X 253.756,Y -140.385,Z 121.324,A 151.047,B 90.000,C 0.000} C_DIS
LIN {X 253.953,Y -140.028,Z 121.281,A 151.128,B 90.000,C 0.000} C_DIS
LIN {X 254.035,Y -139.879,Z 121.179,A 151.162,B 90.000,C 0.000} C_DIS
LIN {X 254.232,Y -139.521,Z 121.137,A 151.242,B 90.000,C 0.000} C_DIS
LIN {X 254.273,Y -139.447,Z 121.085,A 151.259,B 90.000,C 0.000} C_DIS
LIN {X 254.303,Y -139.391,Z 121.034,A 151.272,B 90.000,C 0.000} C_DIS
LIN {X 254.450,Y -139.123,Z 120.992,A 151.332,B 90.000,C 0.000} C_DIS
LIN {X 254.481,Y -139.067,Z 120.941,A 151.345,B 90.000,C 0.000} C_DIS
LIN {X 254.521,Y -138.992,Z 120.890,A 151.361,B 90.000,C 0.000} C_DIS
LIN {X 254.717,Y -138.634,Z 120.847,A 151.442,B 90.000,C 0.000} C_DIS
LIN {X 254.757,Y -138.559,Z 120.796,A 151.459,B 90.000,C 0.000} C_DIS
LIN {X 254.788,Y -138.503,Z 120.745,A 151.471,B 90.000,C 0.000} C_DIS
LIN {X 254.934,Y -138.234,Z 120.703,A 151.532,B 90.000,C 0.000} C_DIS
LIN {X 254.964,Y -138.178,Z 120.652,A 151.544,B 90.000,C 0.000} C_DIS
LIN {X 255.005,Y -138.103,Z 120.601,A 151.561,B 90.000,C 0.000} C_DIS
LIN {X 255.199,Y -137.744,Z 120.558,A 151.642,B 90.000,C 0.000} C_DIS
LIN {X 255.280,Y -137.595,Z 120.456,A 151.675,B 90.000,C 0.000} C_DIS
LIN {X 255.473,Y -137.235,Z 120.414,A 151.756,B 90.000,C 0.000} C_DIS
LIN {X 255.513,Y -137.160,Z 120.363,A 151.773,B 90.000,C 0.000} C_DIS
LIN {X 255.543,Y -137.104,Z 120.312,A 151.786,B 90.000,C 0.000} C_DIS
LIN {X 255.688,Y -136.834,Z 120.269,A 151.846,B 90.000,C 0.000} C_DIS
LIN {X 255.718,Y -136.778,Z 120.218,A 151.859,B 90.000,C 0.000} C_DIS
LIN {X 255.758,Y -136.703,Z 120.167,A 151.875,B 90.000,C 0.000} C_DIS
LIN {X 255.950,Y -136.343,Z 120.125,A 151.956,B 90.000,C 0.000} C_DIS
LIN {X 256.030,Y -136.193,Z 120.023,A 151.990,B 90.000,C 0.000} C_DIS
LIN {X 256.222,Y -135.833,Z 119.980,A 152.070,B 90.000,C 0.000} C_DIS
LIN {X 256.261,Y -135.758,Z 119.929,A 152.087,B 90.000,C 0.000} C_DIS
LIN {X 256.291,Y -135.701,Z 119.878,A 152.100,B 90.000,C 0.000} C_DIS
LIN {X 256.434,Y -135.431,Z 119.836,A 152.160,B 90.000,C 0.000} C_DIS
LIN {X 256.464,Y -135.374,Z 119.785,A 152.173,B 90.000,C 0.000} C_DIS
LIN {X 256.504,Y -135.299,Z 119.734,A 152.189,B 90.000,C 0.000} C_DIS
LIN {X 256.694,Y -134.938,Z 119.691,A 152.270,B 90.000,C 0.000} C_DIS
LIN {X 256.773,Y -134.788,Z 119.589,A 152.304,B 90.000,C 0.000} C_DIS
LIN {X 256.962,Y -134.426,Z 119.547,A 152.384,B 90.000,C 0.000} C_DIS
LIN {X 257.002,Y -134.351,Z 119.496,A 152.401,B 90.000,C 0.000} C_DIS
LIN {X 257.031,Y -134.294,Z 119.445,A 152.414,B 90.000,C 0.000} C_DIS
LIN {X 257.173,Y -134.023,Z 119.402,A 152.474,B 90.000,C 0.000} C_DIS
LIN {X 257.202,Y -133.966,Z 119.351,A 152.487,B 90.000,C 0.000} C_DIS
LIN {X 257.241,Y -133.891,Z 119.300,A 152.504,B 90.000,C 0.000} C_DIS
LIN {X 257.430,Y -133.529,Z 119.258,A 152.584,B 90.000,C 0.000} C_DIS
LIN {X 257.508,Y -133.378,Z 119.156,A 152.618,B 90.000,C 0.000} C_DIS
LIN {X 257.695,Y -133.015,Z 119.113,A 152.698,B 90.000,C 0.000} C_DIS
LIN {X 257.734,Y -132.940,Z 119.062,A 152.715,B 90.000,C 0.000} C_DIS
LIN {X 257.764,Y -132.883,Z 119.011,A 152.728,B 90.000,C 0.000} C_DIS
LIN {X 257.904,Y -132.611,Z 118.969,A 152.788,B 90.000,C 0.000} C_DIS
LIN {X 257.933,Y -132.554,Z 118.918,A 152.801,B 90.000,C 0.000} C_DIS
LIN {X 257.972,Y -132.479,Z 118.867,A 152.818,B 90.000,C 0.000} C_DIS
LIN {X 258.158,Y -132.115,Z 118.824,A 152.898,B 90.000,C 0.000} C_DIS
LIN {X 258.235,Y -131.964,Z 118.722,A 152.932,B 90.000,C 0.000} C_DIS
LIN {X 258.421,Y -131.601,Z 118.680,A 153.013,B 90.000,C 0.000} C_DIS
LIN {X 258.459,Y -131.525,Z 118.629,A 153.029,B 90.000,C 0.000} C_DIS
LIN {X 258.488,Y -131.468,Z 118.577,A 153.042,B 90.000,C 0.000} C_DIS
LIN {X 258.627,Y -131.195,Z 118.535,A 153.102,B 90.000,C 0.000} C_DIS
LIN {X 258.656,Y -131.138,Z 118.484,A 153.115,B 90.000,C 0.000} C_DIS
LIN {X 258.694,Y -131.063,Z 118.433,A 153.132,B 90.000,C 0.000} C_DIS
LIN {X 258.878,Y -130.698,Z 118.390,A 153.212,B 90.000,C 0.000} C_DIS
LIN {X 258.955,Y -130.547,Z 118.288,A 153.246,B 90.000,C 0.000} C_DIS
LIN {X 259.138,Y -130.182,Z 118.246,A 153.327,B 90.000,C 0.000} C_DIS
LIN {X 259.176,Y -130.106,Z 118.195,A 153.343,B 90.000,C 0.000} C_DIS
LIN {X 259.205,Y -130.049,Z 118.144,A 153.356,B 90.000,C 0.000} C_DIS
LIN {X 259.342,Y -129.775,Z 118.101,A 153.417,B 90.000,C 0.000} C_DIS
LIN {X 259.371,Y -129.718,Z 118.050,A 153.429,B 90.000,C 0.000} C_DIS
LIN {X 259.409,Y -129.642,Z 117.999,A 153.446,B 90.000,C 0.000} C_DIS
LIN {X 259.591,Y -129.277,Z 117.957,A 153.527,B 90.000,C 0.000} C_DIS
LIN {X 259.667,Y -129.125,Z 117.855,A 153.560,B 90.000,C 0.000} C_DIS
LIN {X 259.848,Y -128.759,Z 117.812,A 153.641,B 90.000,C 0.000} C_DIS
LIN {X 259.886,Y -128.683,Z 117.761,A 153.658,B 90.000,C 0.000} C_DIS
LIN {X 259.914,Y -128.626,Z 117.710,A 153.670,B 90.000,C 0.000} C_DIS
LIN {X 260.050,Y -128.352,Z 117.668,A 153.731,B 90.000,C 0.000} C_DIS
LIN {X 260.078,Y -128.295,Z 117.617,A 153.743,B 90.000,C 0.000} C_DIS
LIN {X 260.115,Y -128.218,Z 117.566,A 153.760,B 90.000,C 0.000} C_DIS
LIN {X 260.296,Y -127.852,Z 117.523,A 153.841,B 90.000,C 0.000} C_DIS
LIN {X 260.333,Y -127.776,Z 117.472,A 153.857,B 90.000,C 0.000} C_DIS
LIN {X 260.361,Y -127.719,Z 117.421,A 153.870,B 90.000,C 0.000} C_DIS
LIN {X 260.496,Y -127.444,Z 117.379,A 153.931,B 90.000,C 0.000} C_DIS
LIN {X 260.524,Y -127.386,Z 117.328,A 153.943,B 90.000,C 0.000} C_DIS
LIN {X 260.561,Y -127.310,Z 117.277,A 153.960,B 90.000,C 0.000} C_DIS
LIN {X 260.740,Y -126.943,Z 117.234,A 154.041,B 90.000,C 0.000} C_DIS
LIN {X 260.814,Y -126.791,Z 117.132,A 154.074,B 90.000,C 0.000} C_DIS
LIN {X 260.993,Y -126.423,Z 117.090,A 154.155,B 90.000,C 0.000} C_DIS
LIN {X 261.030,Y -126.347,Z 117.039,A 154.172,B 90.000,C 0.000} C_DIS
LIN {X 261.057,Y -126.289,Z 116.988,A 154.184,B 90.000,C 0.000} C_DIS
LIN {X 261.191,Y -126.014,Z 116.945,A 154.245,B 90.000,C 0.000} C_DIS
LIN {X 261.218,Y -125.956,Z 116.894,A 154.257,B 90.000,C 0.000} C_DIS
LIN {X 261.264,Y -125.861,Z 116.843,A 154.278,B 90.000,C 0.000} C_DIS
LIN {X 261.375,Y -125.631,Z 116.822,A 154.329,B 90.000,C 0.000} C_DIS
LIN {X 261.485,Y -125.401,Z 116.843,A 154.379,B 90.000,C 0.000} C_DIS
LIN {X 261.531,Y -125.305,Z 116.894,A 154.400,B 90.000,C 0.000} C_DIS
LIN {X 261.559,Y -125.248,Z 116.945,A 154.413,B 90.000,C 0.000} C_DIS
LIN {X 261.691,Y -124.971,Z 116.988,A 154.473,B 90.000,C 0.000} C_DIS
LIN {X 261.718,Y -124.914,Z 117.039,A 154.486,B 90.000,C 0.000} C_DIS
LIN {X 261.755,Y -124.837,Z 117.090,A 154.502,B 90.000,C 0.000} C_DIS
LIN {X 261.930,Y -124.469,Z 117.132,A 154.583,B 90.000,C 0.000} C_DIS
LIN {X 261.967,Y -124.392,Z 117.183,A 154.600,B 90.000,C 0.000} C_DIS
LIN {X 261.994,Y -124.334,Z 117.234,A 154.612,B 90.000,C 0.000} C_DIS
LIN {X 262.125,Y -124.058,Z 117.277,A 154.673,B 90.000,C 0.000} C_DIS
LIN {X 262.153,Y -124.000,Z 117.328,A 154.686,B 90.000,C 0.000} C_DIS
LIN {X 262.189,Y -123.923,Z 117.379,A 154.702,B 90.000,C 0.000} C_DIS
LIN {X 262.363,Y -123.554,Z 117.421,A 154.783,B 90.000,C 0.000} C_DIS
LIN {X 262.435,Y -123.400,Z 117.523,A 154.817,B 90.000,C 0.000} C_DIS
LIN {X 262.609,Y -123.031,Z 117.566,A 154.897,B 90.000,C 0.000} C_DIS
LIN {X 262.645,Y -122.954,Z 117.617,A 154.914,B 90.000,C 0.000} C_DIS
LIN {X 262.672,Y -122.896,Z 117.668,A 154.927,B 90.000,C 0.000} C_DIS
LIN {X 262.802,Y -122.619,Z 117.710,A 154.987,B 90.000,C 0.000} C_DIS
LIN {X 262.828,Y -122.561,Z 117.761,A 155.000,B 90.000,C 0.000} C_DIS
LIN {X 262.864,Y -122.484,Z 117.812,A 155.016,B 90.000,C 0.000} C_DIS
LIN {X 263.036,Y -122.114,Z 117.855,A 155.097,B 90.000,C 0.000} C_DIS
LIN {X 263.072,Y -122.037,Z 117.906,A 155.114,B 90.000,C 0.000} C_DIS
LIN {X 263.099,Y -121.979,Z 117.957,A 155.126,B 90.000,C 0.000} C_DIS
LIN {X 263.228,Y -121.701,Z 117.999,A 155.187,B 90.000,C 0.000} C_DIS
LIN {X 263.254,Y -121.643,Z 118.050,A 155.199,B 90.000,C 0.000} C_DIS
LIN {X 263.290,Y -121.566,Z 118.101,A 155.216,B 90.000,C 0.000} C_DIS
LIN {X 263.461,Y -121.196,Z 118.144,A 155.297,B 90.000,C 0.000} C_DIS
LIN {X 263.532,Y -121.041,Z 118.246,A 155.330,B 90.000,C 0.000} C_DIS
LIN {X 263.702,Y -120.670,Z 118.288,A 155.411,B 90.000,C 0.000} C_DIS
LIN {X 263.737,Y -120.593,Z 118.339,A 155.428,B 90.000,C 0.000} C_DIS
LIN {X 263.764,Y -120.535,Z 118.390,A 155.441,B 90.000,C 0.000} C_DIS
LIN {X 263.891,Y -120.256,Z 118.433,A 155.501,B 90.000,C 0.000} C_DIS
LIN {X 263.917,Y -120.198,Z 118.484,A 155.514,B 90.000,C 0.000} C_DIS
LIN {X 263.952,Y -120.121,Z 118.535,A 155.530,B 90.000,C 0.000} C_DIS
LIN {X 264.121,Y -119.749,Z 118.577,A 155.611,B 90.000,C 0.000} C_DIS
LIN {X 264.156,Y -119.672,Z 118.629,A 155.628,B 90.000,C 0.000} C_DIS
LIN {X 264.183,Y -119.614,Z 118.680,A 155.640,B 90.000,C 0.000} C_DIS
LIN {X 264.309,Y -119.335,Z 118.722,A 155.701,B 90.000,C 0.000} C_DIS
LIN {X 264.335,Y -119.277,Z 118.773,A 155.713,B 90.000,C 0.000} C_DIS
LIN {X 264.370,Y -119.200,Z 118.824,A 155.730,B 90.000,C 0.000} C_DIS
LIN {X 264.537,Y -118.827,Z 118.867,A 155.811,B 90.000,C 0.000} C_DIS
LIN {X 264.607,Y -118.672,Z 118.969,A 155.844,B 90.000,C 0.000} C_DIS
LIN {X 264.774,Y -118.300,Z 119.011,A 155.925,B 90.000,C 0.000} C_DIS
LIN {X 264.808,Y -118.222,Z 119.062,A 155.942,B 90.000,C 0.000} C_DIS
LIN {X 264.834,Y -118.164,Z 119.113,A 155.954,B 90.000,C 0.000} C_DIS
LIN {X 264.959,Y -117.884,Z 119.156,A 156.015,B 90.000,C 0.000} C_DIS
LIN {X 264.985,Y -117.826,Z 119.207,A 156.028,B 90.000,C 0.000} C_DIS
LIN {X 265.019,Y -117.748,Z 119.258,A 156.044,B 90.000,C 0.000} C_DIS
LIN {X 265.185,Y -117.375,Z 119.300,A 156.125,B 90.000,C 0.000} C_DIS
LIN {X 265.219,Y -117.298,Z 119.351,A 156.142,B 90.000,C 0.000} C_DIS
LIN {X 265.245,Y -117.239,Z 119.402,A 156.154,B 90.000,C 0.000} C_DIS
LIN {X 265.369,Y -116.959,Z 119.445,A 156.215,B 90.000,C 0.000} C_DIS
LIN {X 265.394,Y -116.901,Z 119.496,A 156.227,B 90.000,C 0.000} C_DIS
LIN {X 265.429,Y -116.823,Z 119.547,A 156.244,B 90.000,C 0.000} C_DIS
LIN {X 265.593,Y -116.449,Z 119.589,A 156.325,B 90.000,C 0.000} C_DIS
LIN {X 265.661,Y -116.294,Z 119.691,A 156.358,B 90.000,C 0.000} C_DIS
LIN {X 265.824,Y -115.920,Z 119.734,A 156.439,B 90.000,C 0.000} C_DIS
LIN {X 265.858,Y -115.842,Z 119.785,A 156.456,B 90.000,C 0.000} C_DIS
LIN {X 265.884,Y -115.784,Z 119.836,A 156.468,B 90.000,C 0.000} C_DIS
LIN {X 266.006,Y -115.503,Z 119.878,A 156.529,B 90.000,C 0.000} C_DIS
LIN {X 266.031,Y -115.444,Z 119.929,A 156.542,B 90.000,C 0.000} C_DIS
LIN {X 266.065,Y -115.366,Z 119.980,A 156.558,B 90.000,C 0.000} C_DIS
LIN {X 266.227,Y -114.992,Z 120.023,A 156.639,B 90.000,C 0.000} C_DIS
LIN {X 266.294,Y -114.836,Z 120.125,A 156.673,B 90.000,C 0.000} C_DIS
LIN {X 266.456,Y -114.461,Z 120.167,A 156.753,B 90.000,C 0.000} C_DIS
LIN {X 266.489,Y -114.383,Z 120.218,A 156.770,B 90.000,C 0.000} C_DIS
LIN {X 266.515,Y -114.324,Z 120.269,A 156.783,B 90.000,C 0.000} C_DIS
LIN {X 266.635,Y -114.043,Z 120.312,A 156.843,B 90.000,C 0.000} C_DIS
LIN {X 266.660,Y -113.984,Z 120.363,A 156.856,B 90.000,C 0.000} C_DIS
LIN {X 266.693,Y -113.906,Z 120.414,A 156.872,B 90.000,C 0.000} C_DIS
LIN {X 266.854,Y -113.530,Z 120.456,A 156.953,B 90.000,C 0.000} C_DIS
LIN {X 266.887,Y -113.452,Z 120.507,A 156.970,B 90.000,C 0.000} C_DIS
